            FOR index FROM 1 TO Dim(DoubleQuotation_PtB, 1) DO
                position := DoubleQuotation_PtB{index} * font_size;
                next_target.trans := position; last_index := index;

                MoveJ Offs(next_target, x_offset, y_offset, z_offset),write_speed,fine,Alex_Pen_ABB\WObj:=WorkSurface;
            ENDFOR

            ! Raise pen
            MoveL Offs(next_target, x_offset, y_offset, penup_offset),approach_speed,fine,Alex_Pen_ABB\WObj:=WorkSurface;
        ELSEIF character = "'" THEN
            ! Raise pen to avoid drawing of surface
            position := SingleQuotation_PtA{1} * font_size;
            next_target.trans := position;
            MoveJ Offs(next_target, x_offset, y_offset, penup_offset),approach_speed,fine,Alex_Pen_ABB\WObj:=WorkSurface;

            ! Drop pen
            MoveL Offs(next_target, x_offset, y_offset, z_offset),approach_speed,fine,Alex_Pen_ABB\WObj:=WorkSurface;

            FOR index FROM 1 TO Dim(SingleQuotation_PtA, 1) DO
                position := SingleQuotation_PtA{index} * font_size;
                next_target.trans := position; last_index := index;

                MoveJ Offs(next_target, x_offset, y_offset, z_offset),write_speed,fine,Alex_Pen_ABB\WObj:=WorkSurface;
            ENDFOR

            ! Raise pen
            MoveL Offs(next_target, x_offset, y_offset, penup_offset),approach_speed,fine,Alex_Pen_ABB\WObj:=WorkSurface;
        ELSEIF character = "#" THEN
            ! Raise pen to avoid drawing of surface
            position := HashTag_PtA{1} * font_size;
            next_target.trans := position;
            MoveJ Offs(next_target, x_offset, y_offset, penup_offset),approach_speed,fine,Alex_Pen_ABB\WObj:=WorkSurface;

            ! Drop pen
            MoveL Offs(next_target, x_offset, y_offset, z_offset),approach_speed,fine,Alex_Pen_ABB\WObj:=WorkSurface;

            FOR index FROM 1 TO Dim(HashTag_PtA, 1) DO
                position := HashTag_PtA{index} * font_size;
                next_target.trans := position; last_index := index;

                MoveJ Offs(next_target, x_offset, y_offset, z_offset),write_speed,fine,Alex_Pen_ABB\WObj:=WorkSurface;
            ENDFOR

            ! Raise pen
            MoveL Offs(next_target, x_offset, y_offset, penup_offset),approach_speed,fine,Alex_Pen_ABB\WObj:=WorkSurface;

            ! Raise pen to avoid drawing of surface
            position := HashTag_PtB{1} * font_size;
            next_target.trans := position;
            MoveJ Offs(next_target, x_offset, y_offset, penup_offset),approach_speed,fine,Alex_Pen_ABB\WObj:=WorkSurface;

            ! Drop pen
            MoveL Offs(next_target, x_offset, y_offset, z_offset),approach_speed,fine,Alex_Pen_ABB\WObj:=WorkSurface;

            FOR index FROM 1 TO Dim(HashTag_PtB, 1) DO
                position := HashTag_PtB{index} * font_size;
                next_target.trans := position; last_index := index;

                MoveJ Offs(next_target, x_offset, y_offset, z_offset),write_speed,fine,Alex_Pen_ABB\WObj:=WorkSurface;
            ENDFOR

            ! Raise pen
            MoveL Offs(next_target, x_offset, y_offset, penup_offset),approach_speed,fine,Alex_Pen_ABB\WObj:=WorkSurface;
        ELSEIF character = "$" THEN
            ! Raise pen to avoid drawing of surface
            position := Dollar_PtA{1} * font_size;
            next_target.trans := position;
            MoveJ Offs(next_target, x_offset, y_offset, penup_offset),approach_speed,fine,Alex_Pen_ABB\WObj:=WorkSurface;

            ! Drop pen
            MoveL Offs(next_target, x_offset, y_offset, z_offset),approach_speed,fine,Alex_Pen_ABB\WObj:=WorkSurface;

            FOR index FROM 1 TO Dim(Dollar_PtA, 1) DO
                position := Dollar_PtA{index} * font_size;
                next_target.trans := position; last_index := index;

                MoveJ Offs(next_target, x_offset, y_offset, z_offset),write_speed,fine,Alex_Pen_ABB\WObj:=WorkSurface;
            ENDFOR

            ! Raise pen
            MoveL Offs(next_target, x_offset, y_offset, penup_offset),approach_speed,fine,Alex_Pen_ABB\WObj:=WorkSurface;

            ! Raise pen to avoid drawing of surface
            position := Dollar_PtB{1} * font_size;
            next_target.trans := position;
            MoveJ Offs(next_target, x_offset, y_offset, penup_offset),approach_speed,fine,Alex_Pen_ABB\WObj:=WorkSurface;

            ! Drop pen
            MoveL Offs(next_target, x_offset, y_offset, z_offset),approach_speed,fine,Alex_Pen_ABB\WObj:=WorkSurface;

            FOR index FROM 1 TO Dim(Dollar_PtB, 1) DO
                position := Dollar_PtB{index} * font_size;
                next_target.trans := position; last_index := index;

                MoveJ Offs(next_target, x_offset, y_offset, z_offset),write_speed,fine,Alex_Pen_ABB\WObj:=WorkSurface;
            ENDFOR

            ! Raise pen
            MoveL Offs(next_target, x_offset, y_offset, penup_offset),approach_speed,fine,Alex_Pen_ABB\WObj:=WorkSurface;

            ! Raise pen to avoid drawing of surface
            position := Dollar_PtC{1} * font_size;
            next_target.trans := position;
            MoveJ Offs(next_target, x_offset, y_offset, penup_offset),approach_speed,fine,Alex_Pen_ABB\WObj:=WorkSurface;

            ! Drop pen
            MoveL Offs(next_target, x_offset, y_offset, z_offset),approach_speed,fine,Alex_Pen_ABB\WObj:=WorkSurface;

            FOR index FROM 1 TO Dim(Dollar_PtC, 1) DO
                position := Dollar_PtC{index} * font_size;
                next_target.trans := position; last_index := index;

                MoveJ Offs(next_target, x_offset, y_offset, z_offset),write_speed,fine,Alex_Pen_ABB\WObj:=WorkSurface;
            ENDFOR

            ! Raise pen
            MoveL Offs(next_target, x_offset, y_offset, penup_offset),approach_speed,fine,Alex_Pen_ABB\WObj:=WorkSurface;

            ! Raise pen to avoid drawing of surface
            position := Dollar_PtD{1} * font_size;
            next_target.trans := position;
            MoveJ Offs(next_target, x_offset, y_offset, penup_offset),approach_speed,fine,Alex_Pen_ABB\WObj:=WorkSurface;

            ! Drop pen
            MoveL Offs(next_target, x_offset, y_offset, z_offset),approach_speed,fine,Alex_Pen_ABB\WObj:=WorkSurface;

            FOR index FROM 1 TO Dim(Dollar_PtD, 1) DO
                position := Dollar_PtD{index} * font_size;
                next_target.trans := position; last_index := index;

                MoveJ Offs(next_target, x_offset, y_offset, z_offset),write_speed,fine,Alex_Pen_ABB\WObj:=WorkSurface;
            ENDFOR

            ! Raise pen
            MoveL Offs(next_target, x_offset, y_offset, penup_offset),approach_speed,fine,Alex_Pen_ABB\WObj:=WorkSurface;

            ! Raise pen to avoid drawing of surface
            position := Dollar_PtE{1} * font_size;
            next_target.trans := position;
            MoveJ Offs(next_target, x_offset, y_offset, penup_offset),approach_speed,fine,Alex_Pen_ABB\WObj:=WorkSurface;

            ! Drop pen
            MoveL Offs(next_target, x_offset, y_offset, z_offset),approach_speed,fine,Alex_Pen_ABB\WObj:=WorkSurface;

            FOR index FROM 1 TO Dim(Dollar_PtE, 1) DO
                position := Dollar_PtE{index} * font_size;
                next_target.trans := position; last_index := index;

                MoveJ Offs(next_target, x_offset, y_offset, z_offset),write_speed,fine,Alex_Pen_ABB\WObj:=WorkSurface;
            ENDFOR

            ! Raise pen
            MoveL Offs(next_target, x_offset, y_offset, penup_offset),approach_speed,fine,Alex_Pen_ABB\WObj:=WorkSurface;
        ELSEIF character = "%" THEN
            ! Raise pen to avoid drawing of surface
            position := Percent_PtA{1} * font_size;
            next_target.trans := position;
            MoveJ Offs(next_target, x_offset, y_offset, penup_offset),approach_speed,fine,Alex_Pen_ABB\WObj:=WorkSurface;

            ! Drop pen
            MoveL Offs(next_target, x_offset, y_offset, z_offset),approach_speed,fine,Alex_Pen_ABB\WObj:=WorkSurface;

            FOR index FROM 1 TO Dim(Percent_PtA, 1) DO
                position := Percent_PtA{index} * font_size;
                next_target.trans := position; last_index := index;

                MoveJ Offs(next_target, x_offset, y_offset, z_offset),write_speed,fine,Alex_Pen_ABB\WObj:=WorkSurface;
            ENDFOR

            ! Raise pen
            MoveL Offs(next_target, x_offset, y_offset, penup_offset),approach_speed,fine,Alex_Pen_ABB\WObj:=WorkSurface;

            ! Raise pen to avoid drawing of surface
            position := Percent_PtB{1} * font_size;
            next_target.trans := position;
            MoveJ Offs(next_target, x_offset, y_offset, penup_offset),approach_speed,fine,Alex_Pen_ABB\WObj:=WorkSurface;

            ! Drop pen
            MoveL Offs(next_target, x_offset, y_offset, z_offset),approach_speed,fine,Alex_Pen_ABB\WObj:=WorkSurface;

            FOR index FROM 1 TO Dim(Percent_PtB, 1) DO
                position := Percent_PtB{index} * font_size;
                next_target.trans := position; last_index := index;

                MoveJ Offs(next_target, x_offset, y_offset, z_offset),write_speed,fine,Alex_Pen_ABB\WObj:=WorkSurface;
            ENDFOR

            ! Raise pen
            MoveL Offs(next_target, x_offset, y_offset, penup_offset),approach_speed,fine,Alex_Pen_ABB\WObj:=WorkSurface;

            ! Raise pen to avoid drawing of surface
            position := Percent_PtC{1} * font_size;
            next_target.trans := position;
            MoveJ Offs(next_target, x_offset, y_offset, penup_offset),approach_speed,fine,Alex_Pen_ABB\WObj:=WorkSurface;

            ! Drop pen
            MoveL Offs(next_target, x_offset, y_offset, z_offset),approach_speed,fine,Alex_Pen_ABB\WObj:=WorkSurface;

            FOR index FROM 1 TO Dim(Percent_PtC, 1) DO
                position := Percent_PtC{index} * font_size;
                next_target.trans := position; last_index := index;

                MoveJ Offs(next_target, x_offset, y_offset, z_offset),write_speed,fine,Alex_Pen_ABB\WObj:=WorkSurface;
            ENDFOR

            ! Raise pen
            MoveL Offs(next_target, x_offset, y_offset, penup_offset),approach_speed,fine,Alex_Pen_ABB\WObj:=WorkSurface;

            ! Raise pen to avoid drawing of surface
            position := Percent_PtD{1} * font_size;
            next_target.trans := position;
            MoveJ Offs(next_target, x_offset, y_offset, penup_offset),approach_speed,fine,Alex_Pen_ABB\WObj:=WorkSurface;

            ! Drop pen
            MoveL Offs(next_target, x_offset, y_offset, z_offset),approach_speed,fine,Alex_Pen_ABB\WObj:=WorkSurface;

            FOR index FROM 1 TO Dim(Percent_PtD, 1) DO
                position := Percent_PtD{index} * font_size;
                next_target.trans := position; last_index := index;

                MoveJ Offs(next_target, x_offset, y_offset, z_offset),write_speed,fine,Alex_Pen_ABB\WObj:=WorkSurface;
            ENDFOR

            ! Raise pen
            MoveL Offs(next_target, x_offset, y_offset, penup_offset),approach_speed,fine,Alex_Pen_ABB\WObj:=WorkSurface;
        ELSEIF character = "&" THEN
            ! Raise pen to avoid drawing of surface
            position := Ampersand_PtA{1} * font_size;
            next_target.trans := position;
            MoveJ Offs(next_target, x_offset, y_offset, penup_offset),approach_speed,fine,Alex_Pen_ABB\WObj:=WorkSurface;

            ! Drop pen
            MoveL Offs(next_target, x_offset, y_offset, z_offset),approach_speed,fine,Alex_Pen_ABB\WObj:=WorkSurface;

            FOR index FROM 1 TO Dim(Ampersand_PtA, 1) DO
                position := Ampersand_PtA{index} * font_size;
                next_target.trans := position; last_index := index;

                MoveJ Offs(next_target, x_offset, y_offset, z_offset),write_speed,fine,Alex_Pen_ABB\WObj:=WorkSurface;
            ENDFOR

            ! Raise pen
            MoveL Offs(next_target, x_offset, y_offset, penup_offset),approach_speed,fine,Alex_Pen_ABB\WObj:=WorkSurface;

            ! Raise pen to avoid drawing of surface
            position := Ampersand_PtB{1} * font_size;
            next_target.trans := position;
            MoveJ Offs(next_target, x_offset, y_offset, penup_offset),approach_speed,fine,Alex_Pen_ABB\WObj:=WorkSurface;

            ! Drop pen
            MoveL Offs(next_target, x_offset, y_offset, z_offset),approach_speed,fine,Alex_Pen_ABB\WObj:=WorkSurface;

            FOR index FROM 1 TO Dim(Ampersand_PtB, 1) DO
                position := Ampersand_PtB{index} * font_size;
                next_target.trans := position; last_index := index;

                MoveJ Offs(next_target, x_offset, y_offset, z_offset),write_speed,fine,Alex_Pen_ABB\WObj:=WorkSurface;
            ENDFOR

            ! Raise pen
            MoveL Offs(next_target, x_offset, y_offset, penup_offset),approach_speed,fine,Alex_Pen_ABB\WObj:=WorkSurface;

            ! Raise pen to avoid drawing of surface
            position := Ampersand_PtC{1} * font_size;
            next_target.trans := position;
            MoveJ Offs(next_target, x_offset, y_offset, penup_offset),approach_speed,fine,Alex_Pen_ABB\WObj:=WorkSurface;

            ! Drop pen
            MoveL Offs(next_target, x_offset, y_offset, z_offset),approach_speed,fine,Alex_Pen_ABB\WObj:=WorkSurface;

            FOR index FROM 1 TO Dim(Ampersand_PtC, 1) DO
                position := Ampersand_PtC{index} * font_size;
                next_target.trans := position; last_index := index;

                MoveJ Offs(next_target, x_offset, y_offset, z_offset),write_speed,fine,Alex_Pen_ABB\WObj:=WorkSurface;
            ENDFOR

            ! Raise pen
            MoveL Offs(next_target, x_offset, y_offset, penup_offset),approach_speed,fine,Alex_Pen_ABB\WObj:=WorkSurface;
        ELSEIF character = "(" THEN
            ! Raise pen to avoid drawing of surface
            position := OpenBracket_PtA{1} * font_size;
            next_target.trans := position;
            MoveJ Offs(next_target, x_offset, y_offset, penup_offset),approach_speed,fine,Alex_Pen_ABB\WObj:=WorkSurface;

            ! Drop pen
            MoveL Offs(next_target, x_offset, y_offset, z_offset),approach_speed,fine,Alex_Pen_ABB\WObj:=WorkSurface;

            FOR index FROM 1 TO Dim(OpenBracket_PtA, 1) DO
                position := OpenBracket_PtA{index} * font_size;
                next_target.trans := position; last_index := index;

                MoveJ Offs(next_target, x_offset, y_offset, z_offset),write_speed,fine,Alex_Pen_ABB\WObj:=WorkSurface;
            ENDFOR

            ! Raise pen
            MoveL Offs(next_target, x_offset, y_offset, penup_offset),approach_speed,fine,Alex_Pen_ABB\WObj:=WorkSurface;
        ELSEIF character = ")" THEN
            ! Raise pen to avoid drawing of surface
            position := CloseBracket_PtA{1} * font_size;
            next_target.trans := position;
            MoveJ Offs(next_target, x_offset, y_offset, penup_offset),approach_speed,fine,Alex_Pen_ABB\WObj:=WorkSurface;

            ! Drop pen
            MoveL Offs(next_target, x_offset, y_offset, z_offset),approach_speed,fine,Alex_Pen_ABB\WObj:=WorkSurface;

            FOR index FROM 1 TO Dim(CloseBracket_PtA, 1) DO
                position := CloseBracket_PtA{index} * font_size;
                next_target.trans := position; last_index := index;

                MoveJ Offs(next_target, x_offset, y_offset, z_offset),write_speed,fine,Alex_Pen_ABB\WObj:=WorkSurface;
            ENDFOR

            ! Raise pen
            MoveL Offs(next_target, x_offset, y_offset, penup_offset),approach_speed,fine,Alex_Pen_ABB\WObj:=WorkSurface;
        ELSEIF character = "*" THEN
            ! Raise pen to avoid drawing of surface
            position := Asterisk_PtA{1} * font_size;
            next_target.trans := position;
            MoveJ Offs(next_target, x_offset, y_offset, penup_offset),approach_speed,fine,Alex_Pen_ABB\WObj:=WorkSurface;

            ! Drop pen
            MoveL Offs(next_target, x_offset, y_offset, z_offset),approach_speed,fine,Alex_Pen_ABB\WObj:=WorkSurface;

            FOR index FROM 1 TO Dim(Asterisk_PtA, 1) DO
                position := Asterisk_PtA{index} * font_size;
                next_target.trans := position; last_index := index;

                MoveJ Offs(next_target, x_offset, y_offset, z_offset),write_speed,fine,Alex_Pen_ABB\WObj:=WorkSurface;
            ENDFOR

            ! Raise pen
            MoveL Offs(next_target, x_offset, y_offset, penup_offset),approach_speed,fine,Alex_Pen_ABB\WObj:=WorkSurface;
        ELSEIF character = "+" THEN
            ! Raise pen to avoid drawing of surface
            position := Plus_PtA{1} * font_size;
            next_target.trans := position;
            MoveJ Offs(next_target, x_offset, y_offset, penup_offset),approach_speed,fine,Alex_Pen_ABB\WObj:=WorkSurface;

            ! Drop pen
            MoveL Offs(next_target, x_offset, y_offset, z_offset),approach_speed,fine,Alex_Pen_ABB\WObj:=WorkSurface;

            FOR index FROM 1 TO Dim(Plus_PtA, 1) DO
                position := Plus_PtA{index} * font_size;
                next_target.trans := position; last_index := index;

                MoveJ Offs(next_target, x_offset, y_offset, z_offset),write_speed,fine,Alex_Pen_ABB\WObj:=WorkSurface;
            ENDFOR

            ! Raise pen
            MoveL Offs(next_target, x_offset, y_offset, penup_offset),approach_speed,fine,Alex_Pen_ABB\WObj:=WorkSurface;
        ELSEIF character = "," THEN
            ! Raise pen to avoid drawing of surface
            position := Comma_PtA{1} * font_size;
            next_target.trans := position;
            MoveJ Offs(next_target, x_offset, y_offset, penup_offset),approach_speed,fine,Alex_Pen_ABB\WObj:=WorkSurface;

            ! Drop pen
            MoveL Offs(next_target, x_offset, y_offset, z_offset),approach_speed,fine,Alex_Pen_ABB\WObj:=WorkSurface;

            FOR index FROM 1 TO Dim(Comma_PtA, 1) DO
                position := Comma_PtA{index} * font_size;
                next_target.trans := position; last_index := index;

                MoveJ Offs(next_target, x_offset, y_offset, z_offset),write_speed,fine,Alex_Pen_ABB\WObj:=WorkSurface;
            ENDFOR

            ! Raise pen
            MoveL Offs(next_target, x_offset, y_offset, penup_offset),approach_speed,fine,Alex_Pen_ABB\WObj:=WorkSurface;
        ELSEIF character = "-" THEN
            ! Raise pen to avoid drawing of surface
            position := Minus_PtA{1} * font_size;
            next_target.trans := position;
            MoveJ Offs(next_target, x_offset, y_offset, penup_offset),approach_speed,fine,Alex_Pen_ABB\WObj:=WorkSurface;

            ! Drop pen
            MoveL Offs(next_target, x_offset, y_offset, z_offset),approach_speed,fine,Alex_Pen_ABB\WObj:=WorkSurface;

            FOR index FROM 1 TO Dim(Minus_PtA, 1) DO
                position := Minus_PtA{index} * font_size;
                next_target.trans := position; last_index := index;

                MoveJ Offs(next_target, x_offset, y_offset, z_offset),write_speed,fine,Alex_Pen_ABB\WObj:=WorkSurface;
            ENDFOR

            ! Raise pen
            MoveL Offs(next_target, x_offset, y_offset, penup_offset),approach_speed,fine,Alex_Pen_ABB\WObj:=WorkSurface;
        ELSEIF character = "." THEN
            ! Raise pen to avoid drawing of surface
            position := Fullstop_PtA{1} * font_size;
            next_target.trans := position;
            MoveJ Offs(next_target, x_offset, y_offset, penup_offset),approach_speed,fine,Alex_Pen_ABB\WObj:=WorkSurface;

            ! Drop pen
            MoveL Offs(next_target, x_offset, y_offset, z_offset),approach_speed,fine,Alex_Pen_ABB\WObj:=WorkSurface;

            FOR index FROM 1 TO Dim(Fullstop_PtA, 1) DO
                position := Fullstop_PtA{index} * font_size;
                next_target.trans := position; last_index := index;

                MoveJ Offs(next_target, x_offset, y_offset, z_offset),write_speed,fine,Alex_Pen_ABB\WObj:=WorkSurface;
            ENDFOR

            ! Raise pen
            MoveL Offs(next_target, x_offset, y_offset, penup_offset),approach_speed,fine,Alex_Pen_ABB\WObj:=WorkSurface;
        ELSEIF character = "/" THEN
            ! Raise pen to avoid drawing of surface
            position := ForwardSlash_PtA{1} * font_size;
            next_target.trans := position;
            MoveJ Offs(next_target, x_offset, y_offset, penup_offset),approach_speed,fine,Alex_Pen_ABB\WObj:=WorkSurface;

            ! Drop pen
            MoveL Offs(next_target, x_offset, y_offset, z_offset),approach_speed,fine,Alex_Pen_ABB\WObj:=WorkSurface;

            FOR index FROM 1 TO Dim(ForwardSlash_PtA, 1) DO
                position := ForwardSlash_PtA{index} * font_size;
                next_target.trans := position; last_index := index;

                MoveJ Offs(next_target, x_offset, y_offset, z_offset),write_speed,fine,Alex_Pen_ABB\WObj:=WorkSurface;
            ENDFOR

            ! Raise pen
            MoveL Offs(next_target, x_offset, y_offset, penup_offset),approach_speed,fine,Alex_Pen_ABB\WObj:=WorkSurface;
        ELSEIF character = "0" THEN
            ! Raise pen to avoid drawing of surface
            position := Zero_PtA{1} * font_size;
            next_target.trans := position;
            MoveJ Offs(next_target, x_offset, y_offset, penup_offset),approach_speed,fine,Alex_Pen_ABB\WObj:=WorkSurface;

            ! Drop pen
            MoveL Offs(next_target, x_offset, y_offset, z_offset),approach_speed,fine,Alex_Pen_ABB\WObj:=WorkSurface;

            FOR index FROM 1 TO Dim(Zero_PtA, 1) DO
                position := Zero_PtA{index} * font_size;
                next_target.trans := position; last_index := index;

                MoveJ Offs(next_target, x_offset, y_offset, z_offset),write_speed,fine,Alex_Pen_ABB\WObj:=WorkSurface;
            ENDFOR

            ! Raise pen
            MoveL Offs(next_target, x_offset, y_offset, penup_offset),approach_speed,fine,Alex_Pen_ABB\WObj:=WorkSurface;

            ! Raise pen to avoid drawing of surface
            position := Zero_PtB{1} * font_size;
            next_target.trans := position;
            MoveJ Offs(next_target, x_offset, y_offset, penup_offset),approach_speed,fine,Alex_Pen_ABB\WObj:=WorkSurface;

            ! Drop pen
            MoveL Offs(next_target, x_offset, y_offset, z_offset),approach_speed,fine,Alex_Pen_ABB\WObj:=WorkSurface;

            FOR index FROM 1 TO Dim(Zero_PtB, 1) DO
                position := Zero_PtB{index} * font_size;
                next_target.trans := position; last_index := index;

                MoveJ Offs(next_target, x_offset, y_offset, z_offset),write_speed,fine,Alex_Pen_ABB\WObj:=WorkSurface;
            ENDFOR

            ! Raise pen
            MoveL Offs(next_target, x_offset, y_offset, penup_offset),approach_speed,fine,Alex_Pen_ABB\WObj:=WorkSurface;
        ELSEIF character = "1" THEN
            ! Raise pen to avoid drawing of surface
            position := One_PtA{1} * font_size;
            next_target.trans := position;
            MoveJ Offs(next_target, x_offset, y_offset, penup_offset),approach_speed,fine,Alex_Pen_ABB\WObj:=WorkSurface;

            ! Drop pen
            MoveL Offs(next_target, x_offset, y_offset, z_offset),approach_speed,fine,Alex_Pen_ABB\WObj:=WorkSurface;

            FOR index FROM 1 TO Dim(One_PtA, 1) DO
                position := One_PtA{index} * font_size;
                next_target.trans := position; last_index := index;

                MoveJ Offs(next_target, x_offset, y_offset, z_offset),write_speed,fine,Alex_Pen_ABB\WObj:=WorkSurface;
            ENDFOR

            ! Raise pen
            MoveL Offs(next_target, x_offset, y_offset, penup_offset),approach_speed,fine,Alex_Pen_ABB\WObj:=WorkSurface;
        ELSEIF character = "2" THEN
            ! Raise pen to avoid drawing of surface
            position := Two_PtA{1} * font_size;
            next_target.trans := position;
            MoveJ Offs(next_target, x_offset, y_offset, penup_offset),approach_speed,fine,Alex_Pen_ABB\WObj:=WorkSurface;

            ! Drop pen
            MoveL Offs(next_target, x_offset, y_offset, z_offset),approach_speed,fine,Alex_Pen_ABB\WObj:=WorkSurface;

            FOR index FROM 1 TO Dim(Two_PtA, 1) DO
                position := Two_PtA{index} * font_size;
                next_target.trans := position; last_index := index;

                MoveJ Offs(next_target, x_offset, y_offset, z_offset),write_speed,fine,Alex_Pen_ABB\WObj:=WorkSurface;
            ENDFOR

            ! Raise pen
            MoveL Offs(next_target, x_offset, y_offset, penup_offset),approach_speed,fine,Alex_Pen_ABB\WObj:=WorkSurface;
        ELSEIF character = "3" THEN
            ! Raise pen to avoid drawing of surface
            position := Three_PtA{1} * font_size;
            next_target.trans := position;
            MoveJ Offs(next_target, x_offset, y_offset, penup_offset),approach_speed,fine,Alex_Pen_ABB\WObj:=WorkSurface;

            ! Drop pen
            MoveL Offs(next_target, x_offset, y_offset, z_offset),approach_speed,fine,Alex_Pen_ABB\WObj:=WorkSurface;

            FOR index FROM 1 TO Dim(Three_PtA, 1) DO
                position := Three_PtA{index} * font_size;
                next_target.trans := position; last_index := index;

                MoveJ Offs(next_target, x_offset, y_offset, z_offset),write_speed,fine,Alex_Pen_ABB\WObj:=WorkSurface;
            ENDFOR

            ! Raise pen
            MoveL Offs(next_target, x_offset, y_offset, penup_offset),approach_speed,fine,Alex_Pen_ABB\WObj:=WorkSurface;
        ELSEIF character = "4" THEN
            ! Raise pen to avoid drawing of surface
            position := Four_PtA{1} * font_size;
            next_target.trans := position;
            MoveJ Offs(next_target, x_offset, y_offset, penup_offset),approach_speed,fine,Alex_Pen_ABB\WObj:=WorkSurface;

            ! Drop pen
            MoveL Offs(next_target, x_offset, y_offset, z_offset),approach_speed,fine,Alex_Pen_ABB\WObj:=WorkSurface;

            FOR index FROM 1 TO Dim(Four_PtA, 1) DO
                position := Four_PtA{index} * font_size;
                next_target.trans := position; last_index := index;

                MoveJ Offs(next_target, x_offset, y_offset, z_offset),write_speed,fine,Alex_Pen_ABB\WObj:=WorkSurface;
            ENDFOR

            ! Raise pen
            MoveL Offs(next_target, x_offset, y_offset, penup_offset),approach_speed,fine,Alex_Pen_ABB\WObj:=WorkSurface;

            ! Raise pen to avoid drawing of surface
            position := Four_PtB{1} * font_size;
            next_target.trans := position;
            MoveJ Offs(next_target, x_offset, y_offset, penup_offset),approach_speed,fine,Alex_Pen_ABB\WObj:=WorkSurface;

            ! Drop pen
            MoveL Offs(next_target, x_offset, y_offset, z_offset),approach_speed,fine,Alex_Pen_ABB\WObj:=WorkSurface;

            FOR index FROM 1 TO Dim(Four_PtB, 1) DO
                position := Four_PtB{index} * font_size;
                next_target.trans := position; last_index := index;

                MoveJ Offs(next_target, x_offset, y_offset, z_offset),write_speed,fine,Alex_Pen_ABB\WObj:=WorkSurface;
            ENDFOR

            ! Raise pen
            MoveL Offs(next_target, x_offset, y_offset, penup_offset),approach_speed,fine,Alex_Pen_ABB\WObj:=WorkSurface;
        ELSEIF character = "5" THEN
            ! Raise pen to avoid drawing of surface
            position := Five_PtA{1} * font_size;
            next_target.trans := position;
            MoveJ Offs(next_target, x_offset, y_offset, penup_offset),approach_speed,fine,Alex_Pen_ABB\WObj:=WorkSurface;

            ! Drop pen
            MoveL Offs(next_target, x_offset, y_offset, z_offset),approach_speed,fine,Alex_Pen_ABB\WObj:=WorkSurface;

            FOR index FROM 1 TO Dim(Five_PtA, 1) DO
                position := Five_PtA{index} * font_size;
                next_target.trans := position; last_index := index;

                MoveJ Offs(next_target, x_offset, y_offset, z_offset),write_speed,fine,Alex_Pen_ABB\WObj:=WorkSurface;
            ENDFOR

            ! Raise pen
            MoveL Offs(next_target, x_offset, y_offset, penup_offset),approach_speed,fine,Alex_Pen_ABB\WObj:=WorkSurface;
        ELSEIF character = "6" THEN
            ! Raise pen to avoid drawing of surface
            position := Six_PtA{1} * font_size;
            next_target.trans := position;
            MoveJ Offs(next_target, x_offset, y_offset, penup_offset),approach_speed,fine,Alex_Pen_ABB\WObj:=WorkSurface;

            ! Drop pen
            MoveL Offs(next_target, x_offset, y_offset, z_offset),approach_speed,fine,Alex_Pen_ABB\WObj:=WorkSurface;

            FOR index FROM 1 TO Dim(Six_PtA, 1) DO
                position := Six_PtA{index} * font_size;
                next_target.trans := position; last_index := index;

                MoveJ Offs(next_target, x_offset, y_offset, z_offset),write_speed,fine,Alex_Pen_ABB\WObj:=WorkSurface;
            ENDFOR

            ! Raise pen
            MoveL Offs(next_target, x_offset, y_offset, penup_offset),approach_speed,fine,Alex_Pen_ABB\WObj:=WorkSurface;

            ! Raise pen to avoid drawing of surface
            position := Six_PtB{1} * font_size;
            next_target.trans := position;
            MoveJ Offs(next_target, x_offset, y_offset, penup_offset),approach_speed,fine,Alex_Pen_ABB\WObj:=WorkSurface;

            ! Drop pen
            MoveL Offs(next_target, x_offset, y_offset, z_offset),approach_speed,fine,Alex_Pen_ABB\WObj:=WorkSurface;

            FOR index FROM 1 TO Dim(Six_PtB, 1) DO
                position := Six_PtB{index} * font_size;
                next_target.trans := position; last_index := index;

                MoveJ Offs(next_target, x_offset, y_offset, z_offset),write_speed,fine,Alex_Pen_ABB\WObj:=WorkSurface;
            ENDFOR

            ! Raise pen
            MoveL Offs(next_target, x_offset, y_offset, penup_offset),approach_speed,fine,Alex_Pen_ABB\WObj:=WorkSurface;
        ELSEIF character = "7" THEN
            ! Raise pen to avoid drawing of surface
            position := Seven_PtA{1} * font_size;
            next_target.trans := position;
            MoveJ Offs(next_target, x_offset, y_offset, penup_offset),approach_speed,fine,Alex_Pen_ABB\WObj:=WorkSurface;

            ! Drop pen
            MoveL Offs(next_target, x_offset, y_offset, z_offset),approach_speed,fine,Alex_Pen_ABB\WObj:=WorkSurface;

            FOR index FROM 1 TO Dim(Seven_PtA, 1) DO
                position := Seven_PtA{index} * font_size;
                next_target.trans := position; last_index := index;

                MoveJ Offs(next_target, x_offset, y_offset, z_offset),write_speed,fine,Alex_Pen_ABB\WObj:=WorkSurface;
            ENDFOR

            ! Raise pen
            MoveL Offs(next_target, x_offset, y_offset, penup_offset),approach_speed,fine,Alex_Pen_ABB\WObj:=WorkSurface;
        ELSEIF character = "8" THEN
            ! Raise pen to avoid drawing of surface
            position := Eight_PtA{1} * font_size;
            next_target.trans := position;
            MoveJ Offs(next_target, x_offset, y_offset, penup_offset),approach_speed,fine,Alex_Pen_ABB\WObj:=WorkSurface;

            ! Drop pen
            MoveL Offs(next_target, x_offset, y_offset, z_offset),approach_speed,fine,Alex_Pen_ABB\WObj:=WorkSurface;

            FOR index FROM 1 TO Dim(Eight_PtA, 1) DO
                position := Eight_PtA{index} * font_size;
                next_target.trans := position; last_index := index;

                MoveJ Offs(next_target, x_offset, y_offset, z_offset),write_speed,fine,Alex_Pen_ABB\WObj:=WorkSurface;
            ENDFOR

            ! Raise pen
            MoveL Offs(next_target, x_offset, y_offset, penup_offset),approach_speed,fine,Alex_Pen_ABB\WObj:=WorkSurface;

            ! Raise pen to avoid drawing of surface
            position := Eight_PtB{1} * font_size;
            next_target.trans := position;
            MoveJ Offs(next_target, x_offset, y_offset, penup_offset),approach_speed,fine,Alex_Pen_ABB\WObj:=WorkSurface;

            ! Drop pen
            MoveL Offs(next_target, x_offset, y_offset, z_offset),approach_speed,fine,Alex_Pen_ABB\WObj:=WorkSurface;

            FOR index FROM 1 TO Dim(Eight_PtB, 1) DO
                position := Eight_PtB{index} * font_size;
                next_target.trans := position; last_index := index;

                MoveJ Offs(next_target, x_offset, y_offset, z_offset),write_speed,fine,Alex_Pen_ABB\WObj:=WorkSurface;
            ENDFOR

            ! Raise pen
            MoveL Offs(next_target, x_offset, y_offset, penup_offset),approach_speed,fine,Alex_Pen_ABB\WObj:=WorkSurface;

            ! Raise pen to avoid drawing of surface
            position := Eight_PtC{1} * font_size;
            next_target.trans := position;
            MoveJ Offs(next_target, x_offset, y_offset, penup_offset),approach_speed,fine,Alex_Pen_ABB\WObj:=WorkSurface;

            ! Drop pen
            MoveL Offs(next_target, x_offset, y_offset, z_offset),approach_speed,fine,Alex_Pen_ABB\WObj:=WorkSurface;

            FOR index FROM 1 TO Dim(Eight_PtC, 1) DO
                position := Eight_PtC{index} * font_size;
                next_target.trans := position; last_index := index;

                MoveJ Offs(next_target, x_offset, y_offset, z_offset),write_speed,fine,Alex_Pen_ABB\WObj:=WorkSurface;
            ENDFOR

            ! Raise pen
            MoveL Offs(next_target, x_offset, y_offset, penup_offset),approach_speed,fine,Alex_Pen_ABB\WObj:=WorkSurface;
        ELSEIF character = "9" THEN
            ! Raise pen to avoid drawing of surface
            position := Nine_PtA{1} * font_size;
            next_target.trans := position;
            MoveJ Offs(next_target, x_offset, y_offset, penup_offset),approach_speed,fine,Alex_Pen_ABB\WObj:=WorkSurface;

            ! Drop pen
            MoveL Offs(next_target, x_offset, y_offset, z_offset),approach_speed,fine,Alex_Pen_ABB\WObj:=WorkSurface;

            FOR index FROM 1 TO Dim(Nine_PtA, 1) DO
                position := Nine_PtA{index} * font_size;
                next_target.trans := position; last_index := index;

                MoveJ Offs(next_target, x_offset, y_offset, z_offset),write_speed,fine,Alex_Pen_ABB\WObj:=WorkSurface;
            ENDFOR

            ! Raise pen
            MoveL Offs(next_target, x_offset, y_offset, penup_offset),approach_speed,fine,Alex_Pen_ABB\WObj:=WorkSurface;

            ! Raise pen to avoid drawing of surface
            position := Nine_PtB{1} * font_size;
            next_target.trans := position;
            MoveJ Offs(next_target, x_offset, y_offset, penup_offset),approach_speed,fine,Alex_Pen_ABB\WObj:=WorkSurface;

            ! Drop pen
            MoveL Offs(next_target, x_offset, y_offset, z_offset),approach_speed,fine,Alex_Pen_ABB\WObj:=WorkSurface;

            FOR index FROM 1 TO Dim(Nine_PtB, 1) DO
                position := Nine_PtB{index} * font_size;
                next_target.trans := position; last_index := index;

                MoveJ Offs(next_target, x_offset, y_offset, z_offset),write_speed,fine,Alex_Pen_ABB\WObj:=WorkSurface;
            ENDFOR

            ! Raise pen
            MoveL Offs(next_target, x_offset, y_offset, penup_offset),approach_speed,fine,Alex_Pen_ABB\WObj:=WorkSurface;
        ELSEIF character = ":" THEN
            ! Raise pen to avoid drawing of surface
            position := Colon_PtA{1} * font_size;
            next_target.trans := position;
            MoveJ Offs(next_target, x_offset, y_offset, penup_offset),approach_speed,fine,Alex_Pen_ABB\WObj:=WorkSurface;

            ! Drop pen
            MoveL Offs(next_target, x_offset, y_offset, z_offset),approach_speed,fine,Alex_Pen_ABB\WObj:=WorkSurface;

            FOR index FROM 1 TO Dim(Colon_PtA, 1) DO
                position := Colon_PtA{index} * font_size;
                next_target.trans := position; last_index := index;

                MoveJ Offs(next_target, x_offset, y_offset, z_offset),write_speed,fine,Alex_Pen_ABB\WObj:=WorkSurface;
            ENDFOR

            ! Raise pen
            MoveL Offs(next_target, x_offset, y_offset, penup_offset),approach_speed,fine,Alex_Pen_ABB\WObj:=WorkSurface;

            ! Raise pen to avoid drawing of surface
            position := Colon_PtB{1} * font_size;
            next_target.trans := position;
            MoveJ Offs(next_target, x_offset, y_offset, penup_offset),approach_speed,fine,Alex_Pen_ABB\WObj:=WorkSurface;

            ! Drop pen
            MoveL Offs(next_target, x_offset, y_offset, z_offset),approach_speed,fine,Alex_Pen_ABB\WObj:=WorkSurface;

            FOR index FROM 1 TO Dim(Colon_PtB, 1) DO
                position := Colon_PtB{index} * font_size;
                next_target.trans := position; last_index := index;

                MoveJ Offs(next_target, x_offset, y_offset, z_offset),write_speed,fine,Alex_Pen_ABB\WObj:=WorkSurface;
            ENDFOR

            ! Raise pen
            MoveL Offs(next_target, x_offset, y_offset, penup_offset),approach_speed,fine,Alex_Pen_ABB\WObj:=WorkSurface;
        ELSEIF character = ";" THEN
            ! Raise pen to avoid drawing of surface
            position := SemiColon_PtA{1} * font_size;
            next_target.trans := position;
            MoveJ Offs(next_target, x_offset, y_offset, penup_offset),approach_speed,fine,Alex_Pen_ABB\WObj:=WorkSurface;

            ! Drop pen
            MoveL Offs(next_target, x_offset, y_offset, z_offset),approach_speed,fine,Alex_Pen_ABB\WObj:=WorkSurface;

            FOR index FROM 1 TO Dim(SemiColon_PtA, 1) DO
                position := SemiColon_PtA{index} * font_size;
                next_target.trans := position; last_index := index;

                MoveJ Offs(next_target, x_offset, y_offset, z_offset),write_speed,fine,Alex_Pen_ABB\WObj:=WorkSurface;
            ENDFOR

            ! Raise pen
            MoveL Offs(next_target, x_offset, y_offset, penup_offset),approach_speed,fine,Alex_Pen_ABB\WObj:=WorkSurface;

            ! Raise pen to avoid drawing of surface
            position := SemiColon_PtB{1} * font_size;
            next_target.trans := position;
            MoveJ Offs(next_target, x_offset, y_offset, penup_offset),approach_speed,fine,Alex_Pen_ABB\WObj:=WorkSurface;

            ! Drop pen
            MoveL Offs(next_target, x_offset, y_offset, z_offset),approach_speed,fine,Alex_Pen_ABB\WObj:=WorkSurface;

            FOR index FROM 1 TO Dim(SemiColon_PtB, 1) DO
                position := SemiColon_PtB{index} * font_size;
                next_target.trans := position; last_index := index;

                MoveJ Offs(next_target, x_offset, y_offset, z_offset),write_speed,fine,Alex_Pen_ABB\WObj:=WorkSurface;
            ENDFOR

            ! Raise pen
            MoveL Offs(next_target, x_offset, y_offset, penup_offset),approach_speed,fine,Alex_Pen_ABB\WObj:=WorkSurface;
        ELSEIF character = "<" THEN
            ! Raise pen to avoid drawing of surface
            position := OpenAngleBracket_PtA{1} * font_size;
            next_target.trans := position;
            MoveJ Offs(next_target, x_offset, y_offset, penup_offset),approach_speed,fine,Alex_Pen_ABB\WObj:=WorkSurface;

            ! Drop pen
            MoveL Offs(next_target, x_offset, y_offset, z_offset),approach_speed,fine,Alex_Pen_ABB\WObj:=WorkSurface;

            FOR index FROM 1 TO Dim(OpenAngleBracket_PtA, 1) DO
                position := OpenAngleBracket_PtA{index} * font_size;
                next_target.trans := position; last_index := index;

                MoveJ Offs(next_target, x_offset, y_offset, z_offset),write_speed,fine,Alex_Pen_ABB\WObj:=WorkSurface;
            ENDFOR

            ! Raise pen
            MoveL Offs(next_target, x_offset, y_offset, penup_offset),approach_speed,fine,Alex_Pen_ABB\WObj:=WorkSurface;
        ELSEIF character = ">" THEN
            ! Raise pen to avoid drawing of surface
            position := CloseAngleBracket_PtA{1} * font_size;
            next_target.trans := position;
            MoveJ Offs(next_target, x_offset, y_offset, penup_offset),approach_speed,fine,Alex_Pen_ABB\WObj:=WorkSurface;

            ! Drop pen
            MoveL Offs(next_target, x_offset, y_offset, z_offset),approach_speed,fine,Alex_Pen_ABB\WObj:=WorkSurface;

            FOR index FROM 1 TO Dim(CloseAngleBracket_PtA, 1) DO
                position := CloseAngleBracket_PtA{index} * font_size;
                next_target.trans := position; last_index := index;

                MoveJ Offs(next_target, x_offset, y_offset, z_offset),write_speed,fine,Alex_Pen_ABB\WObj:=WorkSurface;
            ENDFOR

            ! Raise pen
            MoveL Offs(next_target, x_offset, y_offset, penup_offset),approach_speed,fine,Alex_Pen_ABB\WObj:=WorkSurface;
        ELSEIF character = "=" THEN
            ! Raise pen to avoid drawing of surface
            position := Equal_PtA{1} * font_size;
            next_target.trans := position;
            MoveJ Offs(next_target, x_offset, y_offset, penup_offset),approach_speed,fine,Alex_Pen_ABB\WObj:=WorkSurface;

            ! Drop pen
            MoveL Offs(next_target, x_offset, y_offset, z_offset),approach_speed,fine,Alex_Pen_ABB\WObj:=WorkSurface;

            FOR index FROM 1 TO Dim(Equal_PtA, 1) DO
                position := Equal_PtA{index} * font_size;
                next_target.trans := position; last_index := index;

                MoveJ Offs(next_target, x_offset, y_offset, z_offset),write_speed,fine,Alex_Pen_ABB\WObj:=WorkSurface;
            ENDFOR

            ! Raise pen
            MoveL Offs(next_target, x_offset, y_offset, penup_offset),approach_speed,fine,Alex_Pen_ABB\WObj:=WorkSurface;

            ! Raise pen to avoid drawing of surface
            position := Equal_PtB{1} * font_size;
            next_target.trans := position;
            MoveJ Offs(next_target, x_offset, y_offset, penup_offset),approach_speed,fine,Alex_Pen_ABB\WObj:=WorkSurface;

            ! Drop pen
            MoveL Offs(next_target, x_offset, y_offset, z_offset),approach_speed,fine,Alex_Pen_ABB\WObj:=WorkSurface;

            FOR index FROM 1 TO Dim(Equal_PtB, 1) DO
                position := Equal_PtB{index} * font_size;
                next_target.trans := position; last_index := index;

                MoveJ Offs(next_target, x_offset, y_offset, z_offset),write_speed,fine,Alex_Pen_ABB\WObj:=WorkSurface;
            ENDFOR

            ! Raise pen
            MoveL Offs(next_target, x_offset, y_offset, penup_offset),approach_speed,fine,Alex_Pen_ABB\WObj:=WorkSurface;
        ELSEIF character = "?" THEN
            ! Raise pen to avoid drawing of surface
            position := Question_PtA{1} * font_size;
            next_target.trans := position;
            MoveJ Offs(next_target, x_offset, y_offset, penup_offset),approach_speed,fine,Alex_Pen_ABB\WObj:=WorkSurface;

            ! Drop pen
            MoveL Offs(next_target, x_offset, y_offset, z_offset),approach_speed,fine,Alex_Pen_ABB\WObj:=WorkSurface;

            FOR index FROM 1 TO Dim(Question_PtA, 1) DO
                position := Question_PtA{index} * font_size;
                next_target.trans := position; last_index := index;

                MoveJ Offs(next_target, x_offset, y_offset, z_offset),write_speed,fine,Alex_Pen_ABB\WObj:=WorkSurface;
            ENDFOR

            ! Raise pen
            MoveL Offs(next_target, x_offset, y_offset, penup_offset),approach_speed,fine,Alex_Pen_ABB\WObj:=WorkSurface;

            ! Raise pen to avoid drawing of surface
            position := Question_PtB{1} * font_size;
            next_target.trans := position;
            MoveJ Offs(next_target, x_offset, y_offset, penup_offset),approach_speed,fine,Alex_Pen_ABB\WObj:=WorkSurface;

            ! Drop pen
            MoveL Offs(next_target, x_offset, y_offset, z_offset),approach_speed,fine,Alex_Pen_ABB\WObj:=WorkSurface;

            FOR index FROM 1 TO Dim(Question_PtB, 1) DO
                position := Question_PtB{index} * font_size;
                next_target.trans := position; last_index := index;

                MoveJ Offs(next_target, x_offset, y_offset, z_offset),write_speed,fine,Alex_Pen_ABB\WObj:=WorkSurface;
            ENDFOR

            ! Raise pen
            MoveL Offs(next_target, x_offset, y_offset, penup_offset),approach_speed,fine,Alex_Pen_ABB\WObj:=WorkSurface;
        ELSEIF character = "@" THEN
            ! Raise pen to avoid drawing of surface
            position := At_PtA{1} * font_size;
            next_target.trans := position;
            MoveJ Offs(next_target, x_offset, y_offset, penup_offset),approach_speed,fine,Alex_Pen_ABB\WObj:=WorkSurface;

            ! Drop pen
            MoveL Offs(next_target, x_offset, y_offset, z_offset),approach_speed,fine,Alex_Pen_ABB\WObj:=WorkSurface;

            FOR index FROM 1 TO Dim(At_PtA, 1) DO
                position := At_PtA{index} * font_size;
                next_target.trans := position; last_index := index;

                MoveJ Offs(next_target, x_offset, y_offset, z_offset),write_speed,fine,Alex_Pen_ABB\WObj:=WorkSurface;
            ENDFOR

            ! Raise pen
            MoveL Offs(next_target, x_offset, y_offset, penup_offset),approach_speed,fine,Alex_Pen_ABB\WObj:=WorkSurface;

            ! Raise pen to avoid drawing of surface
            position := At_PtB{1} * font_size;
            next_target.trans := position;
            MoveJ Offs(next_target, x_offset, y_offset, penup_offset),approach_speed,fine,Alex_Pen_ABB\WObj:=WorkSurface;

            ! Drop pen
            MoveL Offs(next_target, x_offset, y_offset, z_offset),approach_speed,fine,Alex_Pen_ABB\WObj:=WorkSurface;

            FOR index FROM 1 TO Dim(At_PtB, 1) DO
                position := At_PtB{index} * font_size;
                next_target.trans := position; last_index := index;

                MoveJ Offs(next_target, x_offset, y_offset, z_offset),write_speed,fine,Alex_Pen_ABB\WObj:=WorkSurface;
            ENDFOR

            ! Raise pen
            MoveL Offs(next_target, x_offset, y_offset, penup_offset),approach_speed,fine,Alex_Pen_ABB\WObj:=WorkSurface;

            ! Raise pen to avoid drawing of surface
            position := At_PtC{1} * font_size;
            next_target.trans := position;
            MoveJ Offs(next_target, x_offset, y_offset, penup_offset),approach_speed,fine,Alex_Pen_ABB\WObj:=WorkSurface;

            ! Drop pen
            MoveL Offs(next_target, x_offset, y_offset, z_offset),approach_speed,fine,Alex_Pen_ABB\WObj:=WorkSurface;

            FOR index FROM 1 TO Dim(At_PtC, 1) DO
                position := At_PtC{index} * font_size;
                next_target.trans := position; last_index := index;

                MoveJ Offs(next_target, x_offset, y_offset, z_offset),write_speed,fine,Alex_Pen_ABB\WObj:=WorkSurface;
            ENDFOR

            ! Raise pen
            MoveL Offs(next_target, x_offset, y_offset, penup_offset),approach_speed,fine,Alex_Pen_ABB\WObj:=WorkSurface;

            ! Raise pen to avoid drawing of surface
            position := At_PtD{1} * font_size;
            next_target.trans := position;
            MoveJ Offs(next_target, x_offset, y_offset, penup_offset),approach_speed,fine,Alex_Pen_ABB\WObj:=WorkSurface;

            ! Drop pen
            MoveL Offs(next_target, x_offset, y_offset, z_offset),approach_speed,fine,Alex_Pen_ABB\WObj:=WorkSurface;

            FOR index FROM 1 TO Dim(At_PtD, 1) DO
                position := At_PtD{index} * font_size;
                next_target.trans := position; last_index := index;

                MoveJ Offs(next_target, x_offset, y_offset, z_offset),write_speed,fine,Alex_Pen_ABB\WObj:=WorkSurface;
            ENDFOR

            ! Raise pen
            MoveL Offs(next_target, x_offset, y_offset, penup_offset),approach_speed,fine,Alex_Pen_ABB\WObj:=WorkSurface;

            ! Raise pen to avoid drawing of surface
            position := At_PtE{1} * font_size;
            next_target.trans := position;
            MoveJ Offs(next_target, x_offset, y_offset, penup_offset),approach_speed,fine,Alex_Pen_ABB\WObj:=WorkSurface;

            ! Drop pen
            MoveL Offs(next_target, x_offset, y_offset, z_offset),approach_speed,fine,Alex_Pen_ABB\WObj:=WorkSurface;

            FOR index FROM 1 TO Dim(At_PtE, 1) DO
                position := At_PtE{index} * font_size;
                next_target.trans := position; last_index := index;

                MoveJ Offs(next_target, x_offset, y_offset, z_offset),write_speed,fine,Alex_Pen_ABB\WObj:=WorkSurface;
            ENDFOR

            ! Raise pen
            MoveL Offs(next_target, x_offset, y_offset, penup_offset),approach_speed,fine,Alex_Pen_ABB\WObj:=WorkSurface;
        ELSEIF character = "A" THEN
            ! Raise pen to avoid drawing of surface
            position := Upper_A_PtA{1} * font_size;
            next_target.trans := position;
            MoveJ Offs(next_target, x_offset, y_offset, penup_offset),approach_speed,fine,Alex_Pen_ABB\WObj:=WorkSurface;

            ! Drop pen
            MoveL Offs(next_target, x_offset, y_offset, z_offset),approach_speed,fine,Alex_Pen_ABB\WObj:=WorkSurface;

            FOR index FROM 1 TO Dim(Upper_A_PtA, 1) DO
                position := Upper_A_PtA{index} * font_size;
                next_target.trans := position; last_index := index;

                MoveJ Offs(next_target, x_offset, y_offset, z_offset),write_speed,fine,Alex_Pen_ABB\WObj:=WorkSurface;
            ENDFOR

            ! Raise pen
            MoveL Offs(next_target, x_offset, y_offset, penup_offset),approach_speed,fine,Alex_Pen_ABB\WObj:=WorkSurface;

            ! Raise pen to avoid drawing of surface
            position := Upper_A_PtB{1} * font_size;
            next_target.trans := position;
            MoveJ Offs(next_target, x_offset, y_offset, penup_offset),approach_speed,fine,Alex_Pen_ABB\WObj:=WorkSurface;

            ! Drop pen
            MoveL Offs(next_target, x_offset, y_offset, z_offset),approach_speed,fine,Alex_Pen_ABB\WObj:=WorkSurface;

            FOR index FROM 1 TO Dim(Upper_A_PtB, 1) DO
                position := Upper_A_PtB{index} * font_size;
                next_target.trans := position; last_index := index;

                MoveJ Offs(next_target, x_offset, y_offset, z_offset),write_speed,fine,Alex_Pen_ABB\WObj:=WorkSurface;
            ENDFOR

            ! Raise pen
            MoveL Offs(next_target, x_offset, y_offset, penup_offset),approach_speed,fine,Alex_Pen_ABB\WObj:=WorkSurface;
        ELSEIF character = "B" THEN
            ! Raise pen to avoid drawing of surface
            position := Upper_B_PtA{1} * font_size;
            next_target.trans := position;
            MoveJ Offs(next_target, x_offset, y_offset, penup_offset),approach_speed,fine,Alex_Pen_ABB\WObj:=WorkSurface;

            ! Drop pen
            MoveL Offs(next_target, x_offset, y_offset, z_offset),approach_speed,fine,Alex_Pen_ABB\WObj:=WorkSurface;

            FOR index FROM 1 TO Dim(Upper_B_PtA, 1) DO
                position := Upper_B_PtA{index} * font_size;
                next_target.trans := position; last_index := index;

                MoveJ Offs(next_target, x_offset, y_offset, z_offset),write_speed,fine,Alex_Pen_ABB\WObj:=WorkSurface;
            ENDFOR

            ! Raise pen
            MoveL Offs(next_target, x_offset, y_offset, penup_offset),approach_speed,fine,Alex_Pen_ABB\WObj:=WorkSurface;

            ! Raise pen to avoid drawing of surface
            position := Upper_B_PtB{1} * font_size;
            next_target.trans := position;
            MoveJ Offs(next_target, x_offset, y_offset, penup_offset),approach_speed,fine,Alex_Pen_ABB\WObj:=WorkSurface;

            ! Drop pen
            MoveL Offs(next_target, x_offset, y_offset, z_offset),approach_speed,fine,Alex_Pen_ABB\WObj:=WorkSurface;

            FOR index FROM 1 TO Dim(Upper_B_PtB, 1) DO
                position := Upper_B_PtB{index} * font_size;
                next_target.trans := position; last_index := index;

                MoveJ Offs(next_target, x_offset, y_offset, z_offset),write_speed,fine,Alex_Pen_ABB\WObj:=WorkSurface;
            ENDFOR

            ! Raise pen
            MoveL Offs(next_target, x_offset, y_offset, penup_offset),approach_speed,fine,Alex_Pen_ABB\WObj:=WorkSurface;

            ! Raise pen to avoid drawing of surface
            position := Upper_B_PtC{1} * font_size;
            next_target.trans := position;
            MoveJ Offs(next_target, x_offset, y_offset, penup_offset),approach_speed,fine,Alex_Pen_ABB\WObj:=WorkSurface;

            ! Drop pen
            MoveL Offs(next_target, x_offset, y_offset, z_offset),approach_speed,fine,Alex_Pen_ABB\WObj:=WorkSurface;

            FOR index FROM 1 TO Dim(Upper_B_PtC, 1) DO
                position := Upper_B_PtC{index} * font_size;
                next_target.trans := position; last_index := index;

                MoveJ Offs(next_target, x_offset, y_offset, z_offset),write_speed,fine,Alex_Pen_ABB\WObj:=WorkSurface;
            ENDFOR

            ! Raise pen
            MoveL Offs(next_target, x_offset, y_offset, penup_offset),approach_speed,fine,Alex_Pen_ABB\WObj:=WorkSurface;
        ELSEIF character = "C" THEN
            ! Raise pen to avoid drawing of surface
            position := Upper_C_PtA{1} * font_size;
            next_target.trans := position;
            MoveJ Offs(next_target, x_offset, y_offset, penup_offset),approach_speed,fine,Alex_Pen_ABB\WObj:=WorkSurface;

            ! Drop pen
            MoveL Offs(next_target, x_offset, y_offset, z_offset),approach_speed,fine,Alex_Pen_ABB\WObj:=WorkSurface;

            FOR index FROM 1 TO Dim(Upper_C_PtA, 1) DO
                position := Upper_C_PtA{index} * font_size;
                next_target.trans := position; last_index := index;

                MoveJ Offs(next_target, x_offset, y_offset, z_offset),write_speed,fine,Alex_Pen_ABB\WObj:=WorkSurface;
            ENDFOR

            ! Raise pen
            MoveL Offs(next_target, x_offset, y_offset, penup_offset),approach_speed,fine,Alex_Pen_ABB\WObj:=WorkSurface;
        ELSEIF character = "D" THEN
            ! Raise pen to avoid drawing of surface
            position := Upper_D_PtA{1} * font_size;
            next_target.trans := position;
            MoveJ Offs(next_target, x_offset, y_offset, penup_offset),approach_speed,fine,Alex_Pen_ABB\WObj:=WorkSurface;

            ! Drop pen
            MoveL Offs(next_target, x_offset, y_offset, z_offset),approach_speed,fine,Alex_Pen_ABB\WObj:=WorkSurface;

            FOR index FROM 1 TO Dim(Upper_D_PtA, 1) DO
                position := Upper_D_PtA{index} * font_size;
                next_target.trans := position; last_index := index;

                MoveJ Offs(next_target, x_offset, y_offset, z_offset),write_speed,fine,Alex_Pen_ABB\WObj:=WorkSurface;
            ENDFOR

            ! Raise pen
            MoveL Offs(next_target, x_offset, y_offset, penup_offset),approach_speed,fine,Alex_Pen_ABB\WObj:=WorkSurface;

            ! Raise pen to avoid drawing of surface
            position := Upper_D_PtB{1} * font_size;
            next_target.trans := position;
            MoveJ Offs(next_target, x_offset, y_offset, penup_offset),approach_speed,fine,Alex_Pen_ABB\WObj:=WorkSurface;

            ! Drop pen
            MoveL Offs(next_target, x_offset, y_offset, z_offset),approach_speed,fine,Alex_Pen_ABB\WObj:=WorkSurface;

            FOR index FROM 1 TO Dim(Upper_D_PtB, 1) DO
                position := Upper_D_PtB{index} * font_size;
                next_target.trans := position; last_index := index;

                MoveJ Offs(next_target, x_offset, y_offset, z_offset),write_speed,fine,Alex_Pen_ABB\WObj:=WorkSurface;
            ENDFOR

            ! Raise pen
            MoveL Offs(next_target, x_offset, y_offset, penup_offset),approach_speed,fine,Alex_Pen_ABB\WObj:=WorkSurface;
        ELSEIF character = "E" THEN
            ! Raise pen to avoid drawing of surface
            position := Upper_E_PtA{1} * font_size;
            next_target.trans := position;
            MoveJ Offs(next_target, x_offset, y_offset, penup_offset),approach_speed,fine,Alex_Pen_ABB\WObj:=WorkSurface;

            ! Drop pen
            MoveL Offs(next_target, x_offset, y_offset, z_offset),approach_speed,fine,Alex_Pen_ABB\WObj:=WorkSurface;

            FOR index FROM 1 TO Dim(Upper_E_PtA, 1) DO
                position := Upper_E_PtA{index} * font_size;
                next_target.trans := position; last_index := index;

                MoveJ Offs(next_target, x_offset, y_offset, z_offset),write_speed,fine,Alex_Pen_ABB\WObj:=WorkSurface;
            ENDFOR

            ! Raise pen
            MoveL Offs(next_target, x_offset, y_offset, penup_offset),approach_speed,fine,Alex_Pen_ABB\WObj:=WorkSurface;
        ELSEIF character = "F" THEN
            ! Raise pen to avoid drawing of surface
            position := Upper_F_PtA{1} * font_size;
            next_target.trans := position;
            MoveJ Offs(next_target, x_offset, y_offset, penup_offset),approach_speed,fine,Alex_Pen_ABB\WObj:=WorkSurface;

            ! Drop pen
            MoveL Offs(next_target, x_offset, y_offset, z_offset),approach_speed,fine,Alex_Pen_ABB\WObj:=WorkSurface;

            FOR index FROM 1 TO Dim(Upper_F_PtA, 1) DO
                position := Upper_F_PtA{index} * font_size;
                next_target.trans := position; last_index := index;

                MoveJ Offs(next_target, x_offset, y_offset, z_offset),write_speed,fine,Alex_Pen_ABB\WObj:=WorkSurface;
            ENDFOR

            ! Raise pen
            MoveL Offs(next_target, x_offset, y_offset, penup_offset),approach_speed,fine,Alex_Pen_ABB\WObj:=WorkSurface;
        ELSEIF character = "G" THEN
            ! Raise pen to avoid drawing of surface
            position := Upper_G_PtA{1} * font_size;
            next_target.trans := position;
            MoveJ Offs(next_target, x_offset, y_offset, penup_offset),approach_speed,fine,Alex_Pen_ABB\WObj:=WorkSurface;

            ! Drop pen
            MoveL Offs(next_target, x_offset, y_offset, z_offset),approach_speed,fine,Alex_Pen_ABB\WObj:=WorkSurface;

            FOR index FROM 1 TO Dim(Upper_G_PtA, 1) DO
                position := Upper_G_PtA{index} * font_size;
                next_target.trans := position; last_index := index;

                MoveJ Offs(next_target, x_offset, y_offset, z_offset),write_speed,fine,Alex_Pen_ABB\WObj:=WorkSurface;
            ENDFOR

            ! Raise pen
            MoveL Offs(next_target, x_offset, y_offset, penup_offset),approach_speed,fine,Alex_Pen_ABB\WObj:=WorkSurface;
        ELSEIF character = "H" THEN
            ! Raise pen to avoid drawing of surface
            position := Upper_H_PtA{1} * font_size;
            next_target.trans := position;
            MoveJ Offs(next_target, x_offset, y_offset, penup_offset),approach_speed,fine,Alex_Pen_ABB\WObj:=WorkSurface;

            ! Drop pen
            MoveL Offs(next_target, x_offset, y_offset, z_offset),approach_speed,fine,Alex_Pen_ABB\WObj:=WorkSurface;

            FOR index FROM 1 TO Dim(Upper_H_PtA, 1) DO
                position := Upper_H_PtA{index} * font_size;
                next_target.trans := position; last_index := index;

                MoveJ Offs(next_target, x_offset, y_offset, z_offset),write_speed,fine,Alex_Pen_ABB\WObj:=WorkSurface;
            ENDFOR

            ! Raise pen
            MoveL Offs(next_target, x_offset, y_offset, penup_offset),approach_speed,fine,Alex_Pen_ABB\WObj:=WorkSurface;
        ELSEIF character = "I" THEN
            ! Raise pen to avoid drawing of surface
            position := Upper_I_PtA{1} * font_size;
            next_target.trans := position;
            MoveJ Offs(next_target, x_offset, y_offset, penup_offset),approach_speed,fine,Alex_Pen_ABB\WObj:=WorkSurface;

            ! Drop pen
            MoveL Offs(next_target, x_offset, y_offset, z_offset),approach_speed,fine,Alex_Pen_ABB\WObj:=WorkSurface;

            FOR index FROM 1 TO Dim(Upper_I_PtA, 1) DO
                position := Upper_I_PtA{index} * font_size;
                next_target.trans := position; last_index := index;

                MoveJ Offs(next_target, x_offset, y_offset, z_offset),write_speed,fine,Alex_Pen_ABB\WObj:=WorkSurface;
            ENDFOR

            ! Raise pen
            MoveL Offs(next_target, x_offset, y_offset, penup_offset),approach_speed,fine,Alex_Pen_ABB\WObj:=WorkSurface;
        ELSEIF character = "J" THEN
            ! Raise pen to avoid drawing of surface
            position := Upper_J_PtA{1} * font_size;
            next_target.trans := position;
            MoveJ Offs(next_target, x_offset, y_offset, penup_offset),approach_speed,fine,Alex_Pen_ABB\WObj:=WorkSurface;

            ! Drop pen
            MoveL Offs(next_target, x_offset, y_offset, z_offset),approach_speed,fine,Alex_Pen_ABB\WObj:=WorkSurface;

            FOR index FROM 1 TO Dim(Upper_J_PtA, 1) DO
                position := Upper_J_PtA{index} * font_size;
                next_target.trans := position; last_index := index;

                MoveJ Offs(next_target, x_offset, y_offset, z_offset),write_speed,fine,Alex_Pen_ABB\WObj:=WorkSurface;
            ENDFOR

            ! Raise pen
            MoveL Offs(next_target, x_offset, y_offset, penup_offset),approach_speed,fine,Alex_Pen_ABB\WObj:=WorkSurface;
        ELSEIF character = "K" THEN
            ! Raise pen to avoid drawing of surface
            position := Upper_K_PtA{1} * font_size;
            next_target.trans := position;
            MoveJ Offs(next_target, x_offset, y_offset, penup_offset),approach_speed,fine,Alex_Pen_ABB\WObj:=WorkSurface;

            ! Drop pen
            MoveL Offs(next_target, x_offset, y_offset, z_offset),approach_speed,fine,Alex_Pen_ABB\WObj:=WorkSurface;

            FOR index FROM 1 TO Dim(Upper_K_PtA, 1) DO
                position := Upper_K_PtA{index} * font_size;
                next_target.trans := position; last_index := index;

                MoveJ Offs(next_target, x_offset, y_offset, z_offset),write_speed,fine,Alex_Pen_ABB\WObj:=WorkSurface;
            ENDFOR

            ! Raise pen
            MoveL Offs(next_target, x_offset, y_offset, penup_offset),approach_speed,fine,Alex_Pen_ABB\WObj:=WorkSurface;
        ELSEIF character = "L" THEN
            ! Raise pen to avoid drawing of surface
            position := Upper_L_PtA{1} * font_size;
            next_target.trans := position;
            MoveJ Offs(next_target, x_offset, y_offset, penup_offset),approach_speed,fine,Alex_Pen_ABB\WObj:=WorkSurface;

            ! Drop pen
            MoveL Offs(next_target, x_offset, y_offset, z_offset),approach_speed,fine,Alex_Pen_ABB\WObj:=WorkSurface;

            FOR index FROM 1 TO Dim(Upper_L_PtA, 1) DO
                position := Upper_L_PtA{index} * font_size;
                next_target.trans := position; last_index := index;

                MoveJ Offs(next_target, x_offset, y_offset, z_offset),write_speed,fine,Alex_Pen_ABB\WObj:=WorkSurface;
            ENDFOR

            ! Raise pen
            MoveL Offs(next_target, x_offset, y_offset, penup_offset),approach_speed,fine,Alex_Pen_ABB\WObj:=WorkSurface;
        ELSEIF character = "M" THEN
            ! Raise pen to avoid drawing of surface
            position := Upper_M_PtA{1} * font_size;
            next_target.trans := position;
            MoveJ Offs(next_target, x_offset, y_offset, penup_offset),approach_speed,fine,Alex_Pen_ABB\WObj:=WorkSurface;

            ! Drop pen
            MoveL Offs(next_target, x_offset, y_offset, z_offset),approach_speed,fine,Alex_Pen_ABB\WObj:=WorkSurface;

            FOR index FROM 1 TO Dim(Upper_M_PtA, 1) DO
                position := Upper_M_PtA{index} * font_size;
                next_target.trans := position; last_index := index;

                MoveJ Offs(next_target, x_offset, y_offset, z_offset),write_speed,fine,Alex_Pen_ABB\WObj:=WorkSurface;
            ENDFOR

            ! Raise pen
            MoveL Offs(next_target, x_offset, y_offset, penup_offset),approach_speed,fine,Alex_Pen_ABB\WObj:=WorkSurface;
        ELSEIF character = "N" THEN
            ! Raise pen to avoid drawing of surface
            position := Upper_N_PtA{1} * font_size;
            next_target.trans := position;
            MoveJ Offs(next_target, x_offset, y_offset, penup_offset),approach_speed,fine,Alex_Pen_ABB\WObj:=WorkSurface;

            ! Drop pen
            MoveL Offs(next_target, x_offset, y_offset, z_offset),approach_speed,fine,Alex_Pen_ABB\WObj:=WorkSurface;

            FOR index FROM 1 TO Dim(Upper_N_PtA, 1) DO
                position := Upper_N_PtA{index} * font_size;
                next_target.trans := position; last_index := index;

                MoveJ Offs(next_target, x_offset, y_offset, z_offset),write_speed,fine,Alex_Pen_ABB\WObj:=WorkSurface;
            ENDFOR

            ! Raise pen
            MoveL Offs(next_target, x_offset, y_offset, penup_offset),approach_speed,fine,Alex_Pen_ABB\WObj:=WorkSurface;
        ELSEIF character = "O" THEN
            ! Raise pen to avoid drawing of surface
            position := Upper_O_PtA{1} * font_size;
            next_target.trans := position;
            MoveJ Offs(next_target, x_offset, y_offset, penup_offset),approach_speed,fine,Alex_Pen_ABB\WObj:=WorkSurface;

            ! Drop pen
            MoveL Offs(next_target, x_offset, y_offset, z_offset),approach_speed,fine,Alex_Pen_ABB\WObj:=WorkSurface;

            FOR index FROM 1 TO Dim(Upper_O_PtA, 1) DO
                position := Upper_O_PtA{index} * font_size;
                next_target.trans := position; last_index := index;

                MoveJ Offs(next_target, x_offset, y_offset, z_offset),write_speed,fine,Alex_Pen_ABB\WObj:=WorkSurface;
            ENDFOR

            ! Raise pen
            MoveL Offs(next_target, x_offset, y_offset, penup_offset),approach_speed,fine,Alex_Pen_ABB\WObj:=WorkSurface;

            ! Raise pen to avoid drawing of surface
            position := Upper_O_PtB{1} * font_size;
            next_target.trans := position;
            MoveJ Offs(next_target, x_offset, y_offset, penup_offset),approach_speed,fine,Alex_Pen_ABB\WObj:=WorkSurface;

            ! Drop pen
            MoveL Offs(next_target, x_offset, y_offset, z_offset),approach_speed,fine,Alex_Pen_ABB\WObj:=WorkSurface;

            FOR index FROM 1 TO Dim(Upper_O_PtB, 1) DO
                position := Upper_O_PtB{index} * font_size;
                next_target.trans := position; last_index := index;

                MoveJ Offs(next_target, x_offset, y_offset, z_offset),write_speed,fine,Alex_Pen_ABB\WObj:=WorkSurface;
            ENDFOR

            ! Raise pen
            MoveL Offs(next_target, x_offset, y_offset, penup_offset),approach_speed,fine,Alex_Pen_ABB\WObj:=WorkSurface;
        ELSEIF character = "P" THEN
            ! Raise pen to avoid drawing of surface
            position := Upper_P_PtA{1} * font_size;
            next_target.trans := position;
            MoveJ Offs(next_target, x_offset, y_offset, penup_offset),approach_speed,fine,Alex_Pen_ABB\WObj:=WorkSurface;

            ! Drop pen
            MoveL Offs(next_target, x_offset, y_offset, z_offset),approach_speed,fine,Alex_Pen_ABB\WObj:=WorkSurface;

            FOR index FROM 1 TO Dim(Upper_P_PtA, 1) DO
                position := Upper_P_PtA{index} * font_size;
                next_target.trans := position; last_index := index;

                MoveJ Offs(next_target, x_offset, y_offset, z_offset),write_speed,fine,Alex_Pen_ABB\WObj:=WorkSurface;
            ENDFOR

            ! Raise pen
            MoveL Offs(next_target, x_offset, y_offset, penup_offset),approach_speed,fine,Alex_Pen_ABB\WObj:=WorkSurface;

            ! Raise pen to avoid drawing of surface
            position := Upper_P_PtB{1} * font_size;
            next_target.trans := position;
            MoveJ Offs(next_target, x_offset, y_offset, penup_offset),approach_speed,fine,Alex_Pen_ABB\WObj:=WorkSurface;

            ! Drop pen
            MoveL Offs(next_target, x_offset, y_offset, z_offset),approach_speed,fine,Alex_Pen_ABB\WObj:=WorkSurface;

            FOR index FROM 1 TO Dim(Upper_P_PtB, 1) DO
                position := Upper_P_PtB{index} * font_size;
                next_target.trans := position; last_index := index;

                MoveJ Offs(next_target, x_offset, y_offset, z_offset),write_speed,fine,Alex_Pen_ABB\WObj:=WorkSurface;
            ENDFOR

            ! Raise pen
            MoveL Offs(next_target, x_offset, y_offset, penup_offset),approach_speed,fine,Alex_Pen_ABB\WObj:=WorkSurface;
        ELSEIF character = "Q" THEN
            ! Raise pen to avoid drawing of surface
            position := Upper_Q_PtA{1} * font_size;
            next_target.trans := position;
            MoveJ Offs(next_target, x_offset, y_offset, penup_offset),approach_speed,fine,Alex_Pen_ABB\WObj:=WorkSurface;

            ! Drop pen
            MoveL Offs(next_target, x_offset, y_offset, z_offset),approach_speed,fine,Alex_Pen_ABB\WObj:=WorkSurface;

            FOR index FROM 1 TO Dim(Upper_Q_PtA, 1) DO
                position := Upper_Q_PtA{index} * font_size;
                next_target.trans := position; last_index := index;

                MoveJ Offs(next_target, x_offset, y_offset, z_offset),write_speed,fine,Alex_Pen_ABB\WObj:=WorkSurface;
            ENDFOR

            ! Raise pen
            MoveL Offs(next_target, x_offset, y_offset, penup_offset),approach_speed,fine,Alex_Pen_ABB\WObj:=WorkSurface;

            ! Raise pen to avoid drawing of surface
            position := Upper_Q_PtB{1} * font_size;
            next_target.trans := position;
            MoveJ Offs(next_target, x_offset, y_offset, penup_offset),approach_speed,fine,Alex_Pen_ABB\WObj:=WorkSurface;

            ! Drop pen
            MoveL Offs(next_target, x_offset, y_offset, z_offset),approach_speed,fine,Alex_Pen_ABB\WObj:=WorkSurface;

            FOR index FROM 1 TO Dim(Upper_Q_PtB, 1) DO
                position := Upper_Q_PtB{index} * font_size;
                next_target.trans := position; last_index := index;

                MoveJ Offs(next_target, x_offset, y_offset, z_offset),write_speed,fine,Alex_Pen_ABB\WObj:=WorkSurface;
            ENDFOR

            ! Raise pen
            MoveL Offs(next_target, x_offset, y_offset, penup_offset),approach_speed,fine,Alex_Pen_ABB\WObj:=WorkSurface;
        ELSEIF character = "R" THEN
            ! Raise pen to avoid drawing of surface
            position := Upper_R_PtA{1} * font_size;
            next_target.trans := position;
            MoveJ Offs(next_target, x_offset, y_offset, penup_offset),approach_speed,fine,Alex_Pen_ABB\WObj:=WorkSurface;

            ! Drop pen
            MoveL Offs(next_target, x_offset, y_offset, z_offset),approach_speed,fine,Alex_Pen_ABB\WObj:=WorkSurface;

            FOR index FROM 1 TO Dim(Upper_R_PtA, 1) DO
                position := Upper_R_PtA{index} * font_size;
                next_target.trans := position; last_index := index;

                MoveJ Offs(next_target, x_offset, y_offset, z_offset),write_speed,fine,Alex_Pen_ABB\WObj:=WorkSurface;
            ENDFOR

            ! Raise pen
            MoveL Offs(next_target, x_offset, y_offset, penup_offset),approach_speed,fine,Alex_Pen_ABB\WObj:=WorkSurface;

            ! Raise pen to avoid drawing of surface
            position := Upper_R_PtB{1} * font_size;
            next_target.trans := position;
            MoveJ Offs(next_target, x_offset, y_offset, penup_offset),approach_speed,fine,Alex_Pen_ABB\WObj:=WorkSurface;

            ! Drop pen
            MoveL Offs(next_target, x_offset, y_offset, z_offset),approach_speed,fine,Alex_Pen_ABB\WObj:=WorkSurface;

            FOR index FROM 1 TO Dim(Upper_R_PtB, 1) DO
                position := Upper_R_PtB{index} * font_size;
                next_target.trans := position; last_index := index;

                MoveJ Offs(next_target, x_offset, y_offset, z_offset),write_speed,fine,Alex_Pen_ABB\WObj:=WorkSurface;
            ENDFOR

            ! Raise pen
            MoveL Offs(next_target, x_offset, y_offset, penup_offset),approach_speed,fine,Alex_Pen_ABB\WObj:=WorkSurface;
        ELSEIF character = "S" THEN
            ! Raise pen to avoid drawing of surface
            position := Upper_S_PtA{1} * font_size;
            next_target.trans := position;
            MoveJ Offs(next_target, x_offset, y_offset, penup_offset),approach_speed,fine,Alex_Pen_ABB\WObj:=WorkSurface;

            ! Drop pen
            MoveL Offs(next_target, x_offset, y_offset, z_offset),approach_speed,fine,Alex_Pen_ABB\WObj:=WorkSurface;

            FOR index FROM 1 TO Dim(Upper_S_PtA, 1) DO
                position := Upper_S_PtA{index} * font_size;
                next_target.trans := position; last_index := index;

                MoveJ Offs(next_target, x_offset, y_offset, z_offset),write_speed,fine,Alex_Pen_ABB\WObj:=WorkSurface;
            ENDFOR

            ! Raise pen
            MoveL Offs(next_target, x_offset, y_offset, penup_offset),approach_speed,fine,Alex_Pen_ABB\WObj:=WorkSurface;
        ELSEIF character = "T" THEN
            ! Raise pen to avoid drawing of surface
            position := Upper_T_PtA{1} * font_size;
            next_target.trans := position;
            MoveJ Offs(next_target, x_offset, y_offset, penup_offset),approach_speed,fine,Alex_Pen_ABB\WObj:=WorkSurface;

            ! Drop pen
            MoveL Offs(next_target, x_offset, y_offset, z_offset),approach_speed,fine,Alex_Pen_ABB\WObj:=WorkSurface;

            FOR index FROM 1 TO Dim(Upper_T_PtA, 1) DO
                position := Upper_T_PtA{index} * font_size;
                next_target.trans := position; last_index := index;

                MoveJ Offs(next_target, x_offset, y_offset, z_offset),write_speed,fine,Alex_Pen_ABB\WObj:=WorkSurface;
            ENDFOR

            ! Raise pen
            MoveL Offs(next_target, x_offset, y_offset, penup_offset),approach_speed,fine,Alex_Pen_ABB\WObj:=WorkSurface;
        ELSEIF character = "U" THEN
            ! Raise pen to avoid drawing of surface
            position := Upper_U_PtA{1} * font_size;
            next_target.trans := position;
            MoveJ Offs(next_target, x_offset, y_offset, penup_offset),approach_speed,fine,Alex_Pen_ABB\WObj:=WorkSurface;

            ! Drop pen
            MoveL Offs(next_target, x_offset, y_offset, z_offset),approach_speed,fine,Alex_Pen_ABB\WObj:=WorkSurface;

            FOR index FROM 1 TO Dim(Upper_U_PtA, 1) DO
                position := Upper_U_PtA{index} * font_size;
                next_target.trans := position; last_index := index;

                MoveJ Offs(next_target, x_offset, y_offset, z_offset),write_speed,fine,Alex_Pen_ABB\WObj:=WorkSurface;
            ENDFOR

            ! Raise pen
            MoveL Offs(next_target, x_offset, y_offset, penup_offset),approach_speed,fine,Alex_Pen_ABB\WObj:=WorkSurface;
        ELSEIF character = "V" THEN
            ! Raise pen to avoid drawing of surface
            position := Upper_V_PtA{1} * font_size;
            next_target.trans := position;
            MoveJ Offs(next_target, x_offset, y_offset, penup_offset),approach_speed,fine,Alex_Pen_ABB\WObj:=WorkSurface;

            ! Drop pen
            MoveL Offs(next_target, x_offset, y_offset, z_offset),approach_speed,fine,Alex_Pen_ABB\WObj:=WorkSurface;

            FOR index FROM 1 TO Dim(Upper_V_PtA, 1) DO
                position := Upper_V_PtA{index} * font_size;
                next_target.trans := position; last_index := index;

                MoveJ Offs(next_target, x_offset, y_offset, z_offset),write_speed,fine,Alex_Pen_ABB\WObj:=WorkSurface;
            ENDFOR

            ! Raise pen
            MoveL Offs(next_target, x_offset, y_offset, penup_offset),approach_speed,fine,Alex_Pen_ABB\WObj:=WorkSurface;
        ELSEIF character = "W" THEN
            ! Raise pen to avoid drawing of surface
            position := Upper_W_PtA{1} * font_size;
            next_target.trans := position;
            MoveJ Offs(next_target, x_offset, y_offset, penup_offset),approach_speed,fine,Alex_Pen_ABB\WObj:=WorkSurface;

            ! Drop pen
            MoveL Offs(next_target, x_offset, y_offset, z_offset),approach_speed,fine,Alex_Pen_ABB\WObj:=WorkSurface;

            FOR index FROM 1 TO Dim(Upper_W_PtA, 1) DO
                position := Upper_W_PtA{index} * font_size;
                next_target.trans := position; last_index := index;

                MoveJ Offs(next_target, x_offset, y_offset, z_offset),write_speed,fine,Alex_Pen_ABB\WObj:=WorkSurface;
            ENDFOR

            ! Raise pen
            MoveL Offs(next_target, x_offset, y_offset, penup_offset),approach_speed,fine,Alex_Pen_ABB\WObj:=WorkSurface;
        ELSEIF character = "X" THEN
            ! Raise pen to avoid drawing of surface
            position := Upper_X_PtA{1} * font_size;
            next_target.trans := position;
            MoveJ Offs(next_target, x_offset, y_offset, penup_offset),approach_speed,fine,Alex_Pen_ABB\WObj:=WorkSurface;

            ! Drop pen
            MoveL Offs(next_target, x_offset, y_offset, z_offset),approach_speed,fine,Alex_Pen_ABB\WObj:=WorkSurface;

            FOR index FROM 1 TO Dim(Upper_X_PtA, 1) DO
                position := Upper_X_PtA{index} * font_size;
                next_target.trans := position; last_index := index;

                MoveJ Offs(next_target, x_offset, y_offset, z_offset),write_speed,fine,Alex_Pen_ABB\WObj:=WorkSurface;
            ENDFOR

            ! Raise pen
            MoveL Offs(next_target, x_offset, y_offset, penup_offset),approach_speed,fine,Alex_Pen_ABB\WObj:=WorkSurface;
        ELSEIF character = "Y" THEN
            ! Raise pen to avoid drawing of surface
            position := Upper_Y_PtA{1} * font_size;
            next_target.trans := position;
            MoveJ Offs(next_target, x_offset, y_offset, penup_offset),approach_speed,fine,Alex_Pen_ABB\WObj:=WorkSurface;

            ! Drop pen
            MoveL Offs(next_target, x_offset, y_offset, z_offset),approach_speed,fine,Alex_Pen_ABB\WObj:=WorkSurface;

            FOR index FROM 1 TO Dim(Upper_Y_PtA, 1) DO
                position := Upper_Y_PtA{index} * font_size;
                next_target.trans := position; last_index := index;

                MoveJ Offs(next_target, x_offset, y_offset, z_offset),write_speed,fine,Alex_Pen_ABB\WObj:=WorkSurface;
            ENDFOR

            ! Raise pen
            MoveL Offs(next_target, x_offset, y_offset, penup_offset),approach_speed,fine,Alex_Pen_ABB\WObj:=WorkSurface;
        ELSEIF character = "Z" THEN
            ! Raise pen to avoid drawing of surface
            position := Upper_Z_PtA{1} * font_size;
            next_target.trans := position;
            MoveJ Offs(next_target, x_offset, y_offset, penup_offset),approach_speed,fine,Alex_Pen_ABB\WObj:=WorkSurface;

            ! Drop pen
            MoveL Offs(next_target, x_offset, y_offset, z_offset),approach_speed,fine,Alex_Pen_ABB\WObj:=WorkSurface;

            FOR index FROM 1 TO Dim(Upper_Z_PtA, 1) DO
                position := Upper_Z_PtA{index} * font_size;
                next_target.trans := position; last_index := index;

                MoveJ Offs(next_target, x_offset, y_offset, z_offset),write_speed,fine,Alex_Pen_ABB\WObj:=WorkSurface;
            ENDFOR

            ! Raise pen
            MoveL Offs(next_target, x_offset, y_offset, penup_offset),approach_speed,fine,Alex_Pen_ABB\WObj:=WorkSurface;
        ELSEIF character = "[" THEN
            ! Raise pen to avoid drawing of surface
            position := OpenSquareBracket_PtA{1} * font_size;
            next_target.trans := position;
            MoveJ Offs(next_target, x_offset, y_offset, penup_offset),approach_speed,fine,Alex_Pen_ABB\WObj:=WorkSurface;

            ! Drop pen
            MoveL Offs(next_target, x_offset, y_offset, z_offset),approach_speed,fine,Alex_Pen_ABB\WObj:=WorkSurface;

            FOR index FROM 1 TO Dim(OpenSquareBracket_PtA, 1) DO
                position := OpenSquareBracket_PtA{index} * font_size;
                next_target.trans := position; last_index := index;

                MoveJ Offs(next_target, x_offset, y_offset, z_offset),write_speed,fine,Alex_Pen_ABB\WObj:=WorkSurface;
            ENDFOR

            ! Raise pen
            MoveL Offs(next_target, x_offset, y_offset, penup_offset),approach_speed,fine,Alex_Pen_ABB\WObj:=WorkSurface;
        ELSEIF character = "]" THEN
            ! Raise pen to avoid drawing of surface
            position := CloseSquareBracket_PtB{1} * font_size;
            next_target.trans := position;
            MoveJ Offs(next_target, x_offset, y_offset, penup_offset),approach_speed,fine,Alex_Pen_ABB\WObj:=WorkSurface;

            ! Drop pen
            MoveL Offs(next_target, x_offset, y_offset, z_offset),approach_speed,fine,Alex_Pen_ABB\WObj:=WorkSurface;

            FOR index FROM 1 TO Dim(CloseSquareBracket_PtB, 1) DO
                position := CloseSquareBracket_PtB{index} * font_size;
                next_target.trans := position; last_index := index;

                MoveJ Offs(next_target, x_offset, y_offset, z_offset),write_speed,fine,Alex_Pen_ABB\WObj:=WorkSurface;
            ENDFOR

            ! Raise pen
            MoveL Offs(next_target, x_offset, y_offset, penup_offset),approach_speed,fine,Alex_Pen_ABB\WObj:=WorkSurface;
        ELSEIF character = "\\" THEN
            ! Raise pen to avoid drawing of surface
            position := BackSlash_PtA{1} * font_size;
            next_target.trans := position;
            MoveJ Offs(next_target, x_offset, y_offset, penup_offset),approach_speed,fine,Alex_Pen_ABB\WObj:=WorkSurface;

            ! Drop pen
            MoveL Offs(next_target, x_offset, y_offset, z_offset),approach_speed,fine,Alex_Pen_ABB\WObj:=WorkSurface;

            FOR index FROM 1 TO Dim(BackSlash_PtA, 1) DO
                position := BackSlash_PtA{index} * font_size;
                next_target.trans := position; last_index := index;

                MoveJ Offs(next_target, x_offset, y_offset, z_offset),write_speed,fine,Alex_Pen_ABB\WObj:=WorkSurface;
            ENDFOR

            ! Raise pen
            MoveL Offs(next_target, x_offset, y_offset, penup_offset),approach_speed,fine,Alex_Pen_ABB\WObj:=WorkSurface;
        ELSEIF character = "^" THEN
            ! Raise pen to avoid drawing of surface
            position := Power_PtA{1} * font_size;
            next_target.trans := position;
            MoveJ Offs(next_target, x_offset, y_offset, penup_offset),approach_speed,fine,Alex_Pen_ABB\WObj:=WorkSurface;

            ! Drop pen
            MoveL Offs(next_target, x_offset, y_offset, z_offset),approach_speed,fine,Alex_Pen_ABB\WObj:=WorkSurface;

            FOR index FROM 1 TO Dim(Power_PtA, 1) DO
                position := Power_PtA{index} * font_size;
                next_target.trans := position; last_index := index;

                MoveJ Offs(next_target, x_offset, y_offset, z_offset),write_speed,fine,Alex_Pen_ABB\WObj:=WorkSurface;
            ENDFOR

            ! Raise pen
            MoveL Offs(next_target, x_offset, y_offset, penup_offset),approach_speed,fine,Alex_Pen_ABB\WObj:=WorkSurface;
        ELSEIF character = "_" THEN
            ! Raise pen to avoid drawing of surface
            position := Underscore_PtA{1} * font_size;
            next_target.trans := position;
            MoveJ Offs(next_target, x_offset, y_offset, penup_offset),approach_speed,fine,Alex_Pen_ABB\WObj:=WorkSurface;

            ! Drop pen
            MoveL Offs(next_target, x_offset, y_offset, z_offset),approach_speed,fine,Alex_Pen_ABB\WObj:=WorkSurface;

            FOR index FROM 1 TO Dim(Underscore_PtA, 1) DO
                position := Underscore_PtA{index} * font_size;
                next_target.trans := position; last_index := index;

                MoveJ Offs(next_target, x_offset, y_offset, z_offset),write_speed,fine,Alex_Pen_ABB\WObj:=WorkSurface;
            ENDFOR

            ! Raise pen
            MoveL Offs(next_target, x_offset, y_offset, penup_offset),approach_speed,fine,Alex_Pen_ABB\WObj:=WorkSurface;
        ELSEIF character = "`" THEN
            ! Raise pen to avoid drawing of surface
            position := InvertedSingleQuote_PtA{1} * font_size;
            next_target.trans := position;
            MoveJ Offs(next_target, x_offset, y_offset, penup_offset),approach_speed,fine,Alex_Pen_ABB\WObj:=WorkSurface;

            ! Drop pen
            MoveL Offs(next_target, x_offset, y_offset, z_offset),approach_speed,fine,Alex_Pen_ABB\WObj:=WorkSurface;

            FOR index FROM 1 TO Dim(InvertedSingleQuote_PtA, 1) DO
                position := InvertedSingleQuote_PtA{index} * font_size;
                next_target.trans := position; last_index := index;

                MoveJ Offs(next_target, x_offset, y_offset, z_offset),write_speed,fine,Alex_Pen_ABB\WObj:=WorkSurface;
            ENDFOR

            ! Raise pen
            MoveL Offs(next_target, x_offset, y_offset, penup_offset),approach_speed,fine,Alex_Pen_ABB\WObj:=WorkSurface;
        ELSEIF character = "a" THEN
            ! Raise pen to avoid drawing of surface
            position := Lower_A_PtA{1} * font_size;
            next_target.trans := position;
            MoveJ Offs(next_target, x_offset, y_offset, penup_offset),approach_speed,fine,Alex_Pen_ABB\WObj:=WorkSurface;

            ! Drop pen
            MoveL Offs(next_target, x_offset, y_offset, z_offset),approach_speed,fine,Alex_Pen_ABB\WObj:=WorkSurface;

            FOR index FROM 1 TO Dim(Lower_A_PtA, 1) DO
                position := Lower_A_PtA{index} * font_size;
                next_target.trans := position; last_index := index;

                MoveJ Offs(next_target, x_offset, y_offset, z_offset),write_speed,fine,Alex_Pen_ABB\WObj:=WorkSurface;
            ENDFOR

            ! Raise pen
            MoveL Offs(next_target, x_offset, y_offset, penup_offset),approach_speed,fine,Alex_Pen_ABB\WObj:=WorkSurface;

            ! Raise pen to avoid drawing of surface
            position := Lower_A_PtB{1} * font_size;
            next_target.trans := position;
            MoveJ Offs(next_target, x_offset, y_offset, penup_offset),approach_speed,fine,Alex_Pen_ABB\WObj:=WorkSurface;

            ! Drop pen
            MoveL Offs(next_target, x_offset, y_offset, z_offset),approach_speed,fine,Alex_Pen_ABB\WObj:=WorkSurface;

            FOR index FROM 1 TO Dim(Lower_A_PtB, 1) DO
                position := Lower_A_PtB{index} * font_size;
                next_target.trans := position; last_index := index;

                MoveJ Offs(next_target, x_offset, y_offset, z_offset),write_speed,fine,Alex_Pen_ABB\WObj:=WorkSurface;
            ENDFOR

            ! Raise pen
            MoveL Offs(next_target, x_offset, y_offset, penup_offset),approach_speed,fine,Alex_Pen_ABB\WObj:=WorkSurface;
        ELSEIF character = "b" THEN
            ! Raise pen to avoid drawing of surface
            position := Lower_B_PtA{1} * font_size;
            next_target.trans := position;
            MoveJ Offs(next_target, x_offset, y_offset, penup_offset),approach_speed,fine,Alex_Pen_ABB\WObj:=WorkSurface;

            ! Drop pen
            MoveL Offs(next_target, x_offset, y_offset, z_offset),approach_speed,fine,Alex_Pen_ABB\WObj:=WorkSurface;

            FOR index FROM 1 TO Dim(Lower_B_PtA, 1) DO
                position := Lower_B_PtA{index} * font_size;
                next_target.trans := position; last_index := index;

                MoveJ Offs(next_target, x_offset, y_offset, z_offset),write_speed,fine,Alex_Pen_ABB\WObj:=WorkSurface;
            ENDFOR

            ! Raise pen
            MoveL Offs(next_target, x_offset, y_offset, penup_offset),approach_speed,fine,Alex_Pen_ABB\WObj:=WorkSurface;

            ! Raise pen to avoid drawing of surface
            position := Lower_B_PtB{1} * font_size;
            next_target.trans := position;
            MoveJ Offs(next_target, x_offset, y_offset, penup_offset),approach_speed,fine,Alex_Pen_ABB\WObj:=WorkSurface;

            ! Drop pen
            MoveL Offs(next_target, x_offset, y_offset, z_offset),approach_speed,fine,Alex_Pen_ABB\WObj:=WorkSurface;

            FOR index FROM 1 TO Dim(Lower_B_PtB, 1) DO
                position := Lower_B_PtB{index} * font_size;
                next_target.trans := position; last_index := index;

                MoveJ Offs(next_target, x_offset, y_offset, z_offset),write_speed,fine,Alex_Pen_ABB\WObj:=WorkSurface;
            ENDFOR

            ! Raise pen
            MoveL Offs(next_target, x_offset, y_offset, penup_offset),approach_speed,fine,Alex_Pen_ABB\WObj:=WorkSurface;
        ELSEIF character = "c" THEN
            ! Raise pen to avoid drawing of surface
            position := Lower_C_PtA{1} * font_size;
            next_target.trans := position;
            MoveJ Offs(next_target, x_offset, y_offset, penup_offset),approach_speed,fine,Alex_Pen_ABB\WObj:=WorkSurface;

            ! Drop pen
            MoveL Offs(next_target, x_offset, y_offset, z_offset),approach_speed,fine,Alex_Pen_ABB\WObj:=WorkSurface;

            FOR index FROM 1 TO Dim(Lower_C_PtA, 1) DO
                position := Lower_C_PtA{index} * font_size;
                next_target.trans := position; last_index := index;

                MoveJ Offs(next_target, x_offset, y_offset, z_offset),write_speed,fine,Alex_Pen_ABB\WObj:=WorkSurface;
            ENDFOR

            ! Raise pen
            MoveL Offs(next_target, x_offset, y_offset, penup_offset),approach_speed,fine,Alex_Pen_ABB\WObj:=WorkSurface;
        ELSEIF character = "d" THEN
            ! Raise pen to avoid drawing of surface
            position := Lower_D_PtA{1} * font_size;
            next_target.trans := position;
            MoveJ Offs(next_target, x_offset, y_offset, penup_offset),approach_speed,fine,Alex_Pen_ABB\WObj:=WorkSurface;

            ! Drop pen
            MoveL Offs(next_target, x_offset, y_offset, z_offset),approach_speed,fine,Alex_Pen_ABB\WObj:=WorkSurface;

            FOR index FROM 1 TO Dim(Lower_D_PtA, 1) DO
                position := Lower_D_PtA{index} * font_size;
                next_target.trans := position; last_index := index;

                MoveJ Offs(next_target, x_offset, y_offset, z_offset),write_speed,fine,Alex_Pen_ABB\WObj:=WorkSurface;
            ENDFOR

            ! Raise pen
            MoveL Offs(next_target, x_offset, y_offset, penup_offset),approach_speed,fine,Alex_Pen_ABB\WObj:=WorkSurface;

            ! Raise pen to avoid drawing of surface
            position := Lower_D_PtB{1} * font_size;
            next_target.trans := position;
            MoveJ Offs(next_target, x_offset, y_offset, penup_offset),approach_speed,fine,Alex_Pen_ABB\WObj:=WorkSurface;

            ! Drop pen
            MoveL Offs(next_target, x_offset, y_offset, z_offset),approach_speed,fine,Alex_Pen_ABB\WObj:=WorkSurface;

            FOR index FROM 1 TO Dim(Lower_D_PtB, 1) DO
                position := Lower_D_PtB{index} * font_size;
                next_target.trans := position; last_index := index;

                MoveJ Offs(next_target, x_offset, y_offset, z_offset),write_speed,fine,Alex_Pen_ABB\WObj:=WorkSurface;
            ENDFOR

            ! Raise pen
            MoveL Offs(next_target, x_offset, y_offset, penup_offset),approach_speed,fine,Alex_Pen_ABB\WObj:=WorkSurface;
        ELSEIF character = "e" THEN
            ! Raise pen to avoid drawing of surface
            position := Lower_E_PtA{1} * font_size;
            next_target.trans := position;
            MoveJ Offs(next_target, x_offset, y_offset, penup_offset),approach_speed,fine,Alex_Pen_ABB\WObj:=WorkSurface;

            ! Drop pen
            MoveL Offs(next_target, x_offset, y_offset, z_offset),approach_speed,fine,Alex_Pen_ABB\WObj:=WorkSurface;

            FOR index FROM 1 TO Dim(Lower_E_PtA, 1) DO
                position := Lower_E_PtA{index} * font_size;
                next_target.trans := position; last_index := index;

                MoveJ Offs(next_target, x_offset, y_offset, z_offset),write_speed,fine,Alex_Pen_ABB\WObj:=WorkSurface;
            ENDFOR

            ! Raise pen
            MoveL Offs(next_target, x_offset, y_offset, penup_offset),approach_speed,fine,Alex_Pen_ABB\WObj:=WorkSurface;

            ! Raise pen to avoid drawing of surface
            position := Lower_E_PtB{1} * font_size;
            next_target.trans := position;
            MoveJ Offs(next_target, x_offset, y_offset, penup_offset),approach_speed,fine,Alex_Pen_ABB\WObj:=WorkSurface;

            ! Drop pen
            MoveL Offs(next_target, x_offset, y_offset, z_offset),approach_speed,fine,Alex_Pen_ABB\WObj:=WorkSurface;

            FOR index FROM 1 TO Dim(Lower_E_PtB, 1) DO
                position := Lower_E_PtB{index} * font_size;
                next_target.trans := position; last_index := index;

                MoveJ Offs(next_target, x_offset, y_offset, z_offset),write_speed,fine,Alex_Pen_ABB\WObj:=WorkSurface;
            ENDFOR

            ! Raise pen
            MoveL Offs(next_target, x_offset, y_offset, penup_offset),approach_speed,fine,Alex_Pen_ABB\WObj:=WorkSurface;
        ELSEIF character = "f" THEN
            ! Raise pen to avoid drawing of surface
            position := Lower_F_PtA{1} * font_size;
            next_target.trans := position;
            MoveJ Offs(next_target, x_offset, y_offset, penup_offset),approach_speed,fine,Alex_Pen_ABB\WObj:=WorkSurface;

            ! Drop pen
            MoveL Offs(next_target, x_offset, y_offset, z_offset),approach_speed,fine,Alex_Pen_ABB\WObj:=WorkSurface;

            FOR index FROM 1 TO Dim(Lower_F_PtA, 1) DO
                position := Lower_F_PtA{index} * font_size;
                next_target.trans := position; last_index := index;

                MoveJ Offs(next_target, x_offset, y_offset, z_offset),write_speed,fine,Alex_Pen_ABB\WObj:=WorkSurface;
            ENDFOR

            ! Raise pen
            MoveL Offs(next_target, x_offset, y_offset, penup_offset),approach_speed,fine,Alex_Pen_ABB\WObj:=WorkSurface;
        ELSEIF character = "g" THEN
            ! Raise pen to avoid drawing of surface
            position := Lower_G_PtA{1} * font_size;
            next_target.trans := position;
            MoveJ Offs(next_target, x_offset, y_offset, penup_offset),approach_speed,fine,Alex_Pen_ABB\WObj:=WorkSurface;

            ! Drop pen
            MoveL Offs(next_target, x_offset, y_offset, z_offset),approach_speed,fine,Alex_Pen_ABB\WObj:=WorkSurface;

            FOR index FROM 1 TO Dim(Lower_G_PtA, 1) DO
                position := Lower_G_PtA{index} * font_size;
                next_target.trans := position; last_index := index;

                MoveJ Offs(next_target, x_offset, y_offset, z_offset),write_speed,fine,Alex_Pen_ABB\WObj:=WorkSurface;
            ENDFOR

            ! Raise pen
            MoveL Offs(next_target, x_offset, y_offset, penup_offset),approach_speed,fine,Alex_Pen_ABB\WObj:=WorkSurface;

            ! Raise pen to avoid drawing of surface
            position := Lower_G_PtB{1} * font_size;
            next_target.trans := position;
            MoveJ Offs(next_target, x_offset, y_offset, penup_offset),approach_speed,fine,Alex_Pen_ABB\WObj:=WorkSurface;

            ! Drop pen
            MoveL Offs(next_target, x_offset, y_offset, z_offset),approach_speed,fine,Alex_Pen_ABB\WObj:=WorkSurface;

            FOR index FROM 1 TO Dim(Lower_G_PtB, 1) DO
                position := Lower_G_PtB{index} * font_size;
                next_target.trans := position; last_index := index;

                MoveJ Offs(next_target, x_offset, y_offset, z_offset),write_speed,fine,Alex_Pen_ABB\WObj:=WorkSurface;
            ENDFOR

            ! Raise pen
            MoveL Offs(next_target, x_offset, y_offset, penup_offset),approach_speed,fine,Alex_Pen_ABB\WObj:=WorkSurface;
        ELSEIF character = "h" THEN
            ! Raise pen to avoid drawing of surface
            position := Lower_H_PtA{1} * font_size;
            next_target.trans := position;
            MoveJ Offs(next_target, x_offset, y_offset, penup_offset),approach_speed,fine,Alex_Pen_ABB\WObj:=WorkSurface;

            ! Drop pen
            MoveL Offs(next_target, x_offset, y_offset, z_offset),approach_speed,fine,Alex_Pen_ABB\WObj:=WorkSurface;

            FOR index FROM 1 TO Dim(Lower_H_PtA, 1) DO
                position := Lower_H_PtA{index} * font_size;
                next_target.trans := position; last_index := index;

                MoveJ Offs(next_target, x_offset, y_offset, z_offset),write_speed,fine,Alex_Pen_ABB\WObj:=WorkSurface;
            ENDFOR

            ! Raise pen
            MoveL Offs(next_target, x_offset, y_offset, penup_offset),approach_speed,fine,Alex_Pen_ABB\WObj:=WorkSurface;
        ELSEIF character = "i" THEN
            ! Raise pen to avoid drawing of surface
            position := Lower_I_PtA{1} * font_size;
            next_target.trans := position;
            MoveJ Offs(next_target, x_offset, y_offset, penup_offset),approach_speed,fine,Alex_Pen_ABB\WObj:=WorkSurface;

            ! Drop pen
            MoveL Offs(next_target, x_offset, y_offset, z_offset),approach_speed,fine,Alex_Pen_ABB\WObj:=WorkSurface;

            FOR index FROM 1 TO Dim(Lower_I_PtA, 1) DO
                position := Lower_I_PtA{index} * font_size;
                next_target.trans := position; last_index := index;

                MoveJ Offs(next_target, x_offset, y_offset, z_offset),write_speed,fine,Alex_Pen_ABB\WObj:=WorkSurface;
            ENDFOR

            ! Raise pen
            MoveL Offs(next_target, x_offset, y_offset, penup_offset),approach_speed,fine,Alex_Pen_ABB\WObj:=WorkSurface;

            ! Raise pen to avoid drawing of surface
            position := Lower_I_PtB{1} * font_size;
            next_target.trans := position;
            MoveJ Offs(next_target, x_offset, y_offset, penup_offset),approach_speed,fine,Alex_Pen_ABB\WObj:=WorkSurface;

            ! Drop pen
            MoveL Offs(next_target, x_offset, y_offset, z_offset),approach_speed,fine,Alex_Pen_ABB\WObj:=WorkSurface;

            FOR index FROM 1 TO Dim(Lower_I_PtB, 1) DO
                position := Lower_I_PtB{index} * font_size;
                next_target.trans := position; last_index := index;

                MoveJ Offs(next_target, x_offset, y_offset, z_offset),write_speed,fine,Alex_Pen_ABB\WObj:=WorkSurface;
            ENDFOR

            ! Raise pen
            MoveL Offs(next_target, x_offset, y_offset, penup_offset),approach_speed,fine,Alex_Pen_ABB\WObj:=WorkSurface;
        ELSEIF character = "j" THEN
            ! Raise pen to avoid drawing of surface
            position := Lower_J_PtA{1} * font_size;
            next_target.trans := position;
            MoveJ Offs(next_target, x_offset, y_offset, penup_offset),approach_speed,fine,Alex_Pen_ABB\WObj:=WorkSurface;

            ! Drop pen
            MoveL Offs(next_target, x_offset, y_offset, z_offset),approach_speed,fine,Alex_Pen_ABB\WObj:=WorkSurface;

            FOR index FROM 1 TO Dim(Lower_J_PtA, 1) DO
                position := Lower_J_PtA{index} * font_size;
                next_target.trans := position; last_index := index;

                MoveJ Offs(next_target, x_offset, y_offset, z_offset),write_speed,fine,Alex_Pen_ABB\WObj:=WorkSurface;
            ENDFOR

